# B&R Automation Studio project EFI (part 4)

### Cpu.per - X20CP1382/Cpu.per
```iecst
VAR_CONFIG
	gPermanentSN AT %M0; (*Serial Number of the machine*)
	gPermanentVersion AT %M100; (* *)
	gPermanentMachine AT %M148; (* *)
	gPermanentSwBelt AT %M500; (* *)
	gPermanentBlock AT %M600; (* *)
	gPermanentInksParSw AT %M800; (* *)
	gInksPermanentParBar AT %M2000; (* *)
	HoldingRegister AT %MW6000; (* *)
END_VAR
```

### @LIBRARY.LST - X20CP1382/EFI/@LIBRARY.LST
```
Library List, V30
FW;C:\BrAutomation\SafeDESIGNER 4.3\SafePROG\PLC\FW_LIB\PLCopen_SF;PLCopen_SF;3
FW;C:\BrAutomation\SafeDESIGNER 4.3\SafePROG\PLC\SafePCOS_31;SafePCOS_31;0
FW;C:\BrAutomation\SafeDESIGNER 4.3\SafePROG\PLC;IEC;3
```

### BusNavigator.iom - X20CP1382/EFI/BusNavigator.iom
```
IOOffsets (SIBytes=2048, SOBytes=2048, NSIBytes=1024, NSOBytes=1024, ConnectionsValidOffset=24, EMOsOffset=69, EMOsSize=64)
  Module SL1.SM1 (Hardware=X20SL8100, SafeLogicID=1, SafeModuleID=1, SISize=1, SOSize=1, NSISize=132, NSOSize=132, SIOffset=16, SOOffset=12, NSIOffset=0, NSOOffset=0, HWTypeCode=5)
    Channel ExternalMachineOption000 (Mapping=SIX69.0, Variable=SelectMachine)
    Channel BOOL001 (Mapping=NSQX0.0, Variable=g_xInputSelectMachine, SODIndex=0x2580, SODSubIndex=0x1)
    Channel INT001 (Mapping=NSQW2, Variable=ErrorCodeArea1, SODIndex=0x2580, SODSubIndex=0x2)
    Channel INT002 (Mapping=NSQW4, Variable=ErrorCodeArea2, SODIndex=0x2580, SODSubIndex=0x3)
  Module SL1.SM2 (Hardware=X20SC0402, SafeLogicID=1, SafeModuleID=2, SISize=4, SOSize=2, NSISize=1, NSOSize=1, SIOffset=20, SOOffset=16, NSIOffset=132, NSOOffset=132, ConnectionValidBitNumber=0, HWTypeCode=59)
    Channel SafeDigitalInput01 (Mapping=SIX20.0, Variable=InputReset, Address=Cyclic#1.::X20SLX402_006.DInput[1], SODIndex=0x6000, SODSubIndex=0x1)
    Channel SafeDigitalOutput01 (Mapping=SQX16.0, Variable=TransportEnable, SODIndex=0x6200, SODSubIndex=0x1)
    Channel ReleaseOutput01 (Mapping=NSQX132.0, Variable=ReleaseTransport, SODIndex=0x6200, SODSubIndex=0x2)
  Module SL1.SM3 (Hardware=X20SI8110, SafeLogicID=1, SafeModuleID=3, SISize=3, SOSize=0, NSISize=0, NSOSize=0, SIOffset=62, ConnectionValidBitNumber=1, HWTypeCode=27)
    Channel SafeDigitalInput01 (Mapping=SIX62.0, Variable=Rear01EStopBK1, Address=Cyclic#1.::X20SI8110_117.DInput[1], SODIndex=0x6000, SODSubIndex=0x1)
    Channel SafeDigitalInput02 (Mapping=SIX62.1, Variable=Rear02EStopBK1, Address=Cyclic#1.::X20SI8110_117.DInput[2], SODIndex=0x6000, SODSubIndex=0x1)
    Channel SafeDigitalInput03 (Mapping=SIX62.2, Variable=Front01EStopBK1, Address=Cyclic#1.::X20SI8110_117.DInput[3], SODIndex=0x6000, SODSubIndex=0x1)
    Channel SafeDigitalInput04 (Mapping=SIX62.3, Variable=Front02EStopBK1, Address=Cyclic#1.::X20SI8110_117.DInput[4], SODIndex=0x6000, SODSubIndex=0x1)
    Channel SafeDigitalInput05 (Mapping=SIX62.4, Variable=LightCurtain01BK1, Address=Cyclic#1.::X20SI8110_117.DInput[5], SODIndex=0x6000, SODSubIndex=0x1)
    Channel SafeDigitalInput06 (Mapping=SIX62.5, Variable=GuardSwitchBK1, Address=Cyclic#1.::X20SI8110_117.DInput[6], SODIndex=0x6000, SODSubIndex=0x1)
    Channel SafeDigitalInput07 (Mapping=SIX62.6, Variable=LightCurtain02BK1, Address=Cyclic#1.::X20SI8110_117.DInput[7], SODIndex=0x6000, SODSubIndex=0x1)
  Module SL1.SM4 (Hardware=X20SO2110, SafeLogicID=1, SafeModuleID=4, SISize=1, SOSize=1, NSISize=1, NSOSize=1, SIOffset=61, SOOffset=14, NSIOffset=133, NSOOffset=133, ConnectionValidBitNumber=2, HWTypeCode=43)
    Channel SafeDigitalOutput01 (Mapping=SQX14.0, Variable=UpDownBK1Enable, SODIndex=0x6200, SODSubIndex=0x1)
    Channel SafeDigitalOutput02 (Mapping=SQX14.1, Variable=IclaBK1Enable, SODIndex=0x6200, SODSubIndex=0x1)
    Channel ReleaseOutput01 (Mapping=NSQX133.0, Variable=ReleaseUpDownBK1, SODIndex=0x6200, SODSubIndex=0x2)
    Channel ReleaseOutput02 (Mapping=NSQX133.1, Variable=ReleaseIclaBK1, SODIndex=0x6200, SODSubIndex=0x2)
  Module SL1.SM5 (Hardware=X20SI8110, SafeLogicID=1, SafeModuleID=5, SISize=3, SOSize=0, NSISize=0, NSOSize=0, SIOffset=66, ConnectionValidBitNumber=3, HWTypeCode=27)
    Channel SafeDigitalInput01 (Mapping=SIX66.0, Variable=Rear01EStopBK2, Address=Cyclic#1.::X20SI8110_217.DInput[1], SODIndex=0x6000, SODSubIndex=0x1)
    Channel SafeDigitalInput02 (Mapping=SIX66.1, Variable=Rear02EStopBK2, Address=Cyclic#1.::X20SI8110_217.DInput[2], SODIndex=0x6000, SODSubIndex=0x1)
    Channel SafeDigitalInput03 (Mapping=SIX66.2, Variable=Front01EStopBK2, Address=Cyclic#1.::X20SI8110_217.DInput[3], SODIndex=0x6000, SODSubIndex=0x1)
    Channel SafeDigitalInput04 (Mapping=SIX66.3, Variable=Front02EStopBK2, Address=Cyclic#1.::X20SI8110_217.DInput[4], SODIndex=0x6000, SODSubIndex=0x1)
    Channel SafeDigitalInput05 (Mapping=SIX66.4, Variable=LightCurtain01BK2, Address=Cyclic#1.::X20SI8110_217.DInput[5], SODIndex=0x6000, SODSubIndex=0x1)
    Channel SafeDigitalInput06 (Mapping=SIX66.5, Variable=GuardSwitchBK2, Address=Cyclic#1.::X20SI8110_217.DInput[6], SODIndex=0x6000, SODSubIndex=0x1)
    Channel SafeDigitalInput07 (Mapping=SIX66.6, Variable=LightCurtain02BK2, Address=Cyclic#1.::X20SI8110_217.DInput[7], SODIndex=0x6000, SODSubIndex=0x1)
  Module SL1.SM6 (Hardware=X20SO2110, SafeLogicID=1, SafeModuleID=6, SISize=1, SOSize=1, NSISize=1, NSOSize=1, SIOffset=65, SOOffset=15, NSIOffset=134, NSOOffset=134, ConnectionValidBitNumber=4, HWTypeCode=43)
    Channel SafeDigitalOutput01 (Mapping=SQX15.0, Variable=UpDownBK2Enable, SODIndex=0x6200, SODSubIndex=0x1)
    Channel SafeDigitalOutput02 (Mapping=SQX15.1, Variable=IclaBK2Enable, SODIndex=0x6200, SODSubIndex=0x1)
    Channel ReleaseOutput01 (Mapping=NSQX134.0, Variable=ReleaseUpDownBK2, SODIndex=0x6200, SODSubIndex=0x2)
    Channel ReleaseOutput02 (Mapping=NSQX134.1, Variable=ReleaseIclaBK2, SODIndex=0x6200, SODSubIndex=0x2)
```

### CHGUNITS.LST - X20CP1382/EFI/CHGUNITS.LST
```
(*
NPOU: 2
*)
PG	Main
FB	MOVE_UINT
```

### CROSSREF.CSV - X20CP1382/EFI/CROSSREF.CSV
```
C000,POE\Main\Code.GB,4,IN,282,90,Read,,INT,,,VAR_GLOBAL,GLOBAL,,
C000,POE\Main\Code.GB,5,IN,283,55,Read,,INT,,,VAR_GLOBAL,GLOBAL,,
C000,POE\Main\Code.GB,8,IN,287,58,Read,,INT,,,VAR_GLOBAL,GLOBAL,,
C000,POE\Main\Code.GB,8,IN,289,0,Read,,INT,,,VAR_GLOBAL,GLOBAL,,
C000,POE\Main\Code.GB,8,IN,285,39,Read,,INT,,,VAR_GLOBAL,GLOBAL,,
C000,POE\Main\Code.GB,19,IN,421,84,Read,,INT,,,VAR_GLOBAL,GLOBAL,,
C000,POE\Main\Code.GB,20,IN,437,54,Read,,INT,,,VAR_GLOBAL,GLOBAL,,
C000,POE\Main\Code.GB,22,IN,571,82,Read,,INT,,,VAR_GLOBAL,GLOBAL,,
C000,POE\Main\Code.GB,23,IN,493,38,Read,,INT,,,VAR_GLOBAL,GLOBAL,,
C000,POE\Main\Code.GB,23,IN,604,48,Read,,INT,,,VAR_GLOBAL,GLOBAL,,
ErrorCodeArea1,POE\Main\Code.GB,11,OUT,307,71,Write,,INT,NSQW2,,VAR_GLOBAL,GLOBAL,,
ErrorCodeArea2,POE\Main\Code.GB,26,OUT,800,82,Write,,INT,NSQW4,,VAR_GLOBAL,GLOBAL,,
Front01EStopBK1,POE\Main\Code.GB,1,IN,310,8,Read,,SAFEBOOL,SIX62.2,,VAR_GLOBAL,GLOBAL,,
Front01EStopBK2,POE\Main\Code.GB,16,IN,392,8,Read,,SAFEBOOL,SIX66.2,,VAR_GLOBAL,GLOBAL,,
Front02EStopBK1,POE\Main\Code.GB,1,IN,311,8,Read,,SAFEBOOL,SIX62.3,,VAR_GLOBAL,GLOBAL,,
Front02EStopBK2,POE\Main\Code.GB,16,IN,393,8,Read,,SAFEBOOL,SIX66.3,,VAR_GLOBAL,GLOBAL,,
g_xInputSelectMachine,POE\Main\Code.GB,16,OUT,855,37,Write,,BOOL,NSQX0.0,,VAR_GLOBAL,GLOBAL,,
GuardSwitchBK1,POE\Main\Code.GB,4,IN,312,23,Read,,SAFEBOOL,SIX62.5,,VAR_GLOBAL,GLOBAL,,
GuardSwitchBK2,POE\Main\Code.GB,19,IN,477,47,Read,,SAFEBOOL,SIX66.5,,VAR_GLOBAL,GLOBAL,,
IclaBK1Enable,POE\Main\Code.GB,29,OUT,769,81,Write,,SAFEBOOL,SQX14.1,,VAR_GLOBAL,GLOBAL,,
IclaBK2Enable,POE\Main\Code.GB,32,OUT,683,77,Write,,SAFEBOOL,SQX15.1,,VAR_GLOBAL,GLOBAL,,
InputReset,POE\Main\Code.GB,1,IN,37,83,Read,,SAFEBOOL,SIX20.0,,VAR_GLOBAL,GLOBAL,,
InputReset,POE\Main\Code.GB,2,IN,27,0,Read,,SAFEBOOL,SIX20.0,,VAR_GLOBAL,GLOBAL,,
InputReset,POE\Main\Code.GB,7,IN,155,47,Read,,SAFEBOOL,SIX20.0,,VAR_GLOBAL,GLOBAL,,
InputReset,POE\Main\Code.GB,8,IN,211,0,Read,,SAFEBOOL,SIX20.0,,VAR_GLOBAL,GLOBAL,,
InputReset,POE\Main\Code.GB,17,IN,362,30,Read,,SAFEBOOL,SIX20.0,,VAR_GLOBAL,GLOBAL,,
InputReset,POE\Main\Code.GB,20,IN,390,0,Read,,SAFEBOOL,SIX20.0,,VAR_GLOBAL,GLOBAL,,
InputReset,POE\Main\Code.GB,22,IN,547,81,Read,,SAFEBOOL,SIX20.0,,VAR_GLOBAL,GLOBAL,,
InputReset,POE\Main\Code.GB,22,IN,475,58,Read,,SAFEBOOL,SIX20.0,,VAR_GLOBAL,GLOBAL,,
InputReset,POE\Main\Code.GB,29,IN,774,15,Read,,SAFEBOOL,SIX20.0,,VAR_GLOBAL,GLOBAL,,
InputReset,POE\Main\Code.GB,29,IN,718,6,Read,,SAFEBOOL,SIX20.0,,VAR_GLOBAL,GLOBAL,,
InputReset,POE\Main\Code.GB,32,IN,652,23,Read,,SAFEBOOL,SIX20.0,,VAR_GLOBAL,GLOBAL,,
LightCurtain01BK1,POE\Main\Code.GB,7,IN,317,10,Read,,SAFEBOOL,SIX62.4,,VAR_GLOBAL,GLOBAL,,
LightCurtain01BK2,POE\Main\Code.GB,22,IN,549,3,Read,,SAFEBOOL,SIX66.4,,VAR_GLOBAL,GLOBAL,,
LightCurtain02BK1,POE\Main\Code.GB,7,IN,318,9,Read,,SAFEBOOL,SIX62.6,,VAR_GLOBAL,GLOBAL,,
LightCurtain02BK2,POE\Main\Code.GB,22,IN,559,3,Read,,SAFEBOOL,SIX66.6,,VAR_GLOBAL,GLOBAL,,
Rear01EStopBK1,POE\Main\Code.GB,1,IN,308,13,Read,,SAFEBOOL,SIX62.0,,VAR_GLOBAL,GLOBAL,,
Rear01EStopBK2,POE\Main\Code.GB,16,IN,394,49,Read,,SAFEBOOL,SIX66.0,,VAR_GLOBAL,GLOBAL,,
Rear02EStopBK1,POE\Main\Code.GB,1,IN,309,13,Read,,SAFEBOOL,SIX62.1,,VAR_GLOBAL,GLOBAL,,
Rear02EStopBK2,POE\Main\Code.GB,16,IN,395,49,Read,,SAFEBOOL,SIX66.1,,VAR_GLOBAL,GLOBAL,,
ReleaseIclaBK1,POE\Main\Code.GB,30,OUT,773,78,Write,,BOOL,NSQX133.1,,VAR_GLOBAL,GLOBAL,,
ReleaseIclaBK2,POE\Main\Code.GB,33,OUT,689,81,Write,,BOOL,NSQX134.1,,VAR_GLOBAL,GLOBAL,,
ReleaseTransport,POE\Main\Code.GB,27,OUT,719,66,Write,,BOOL,NSQX132.0,,VAR_GLOBAL,GLOBAL,,
ReleaseUpDownBK1,POE\Main\Code.GB,30,OUT,772,74,Write,,BOOL,NSQX133.0,,VAR_GLOBAL,GLOBAL,,
ReleaseUpDownBK2,POE\Main\Code.GB,33,OUT,688,77,Write,,BOOL,NSQX134.0,,VAR_GLOBAL,GLOBAL,,
SelectMachine,POE\Main\Code.GB,16,IN,801,53,Read,,SAFEBOOL,SIX69.0,,VAR_GLOBAL,GLOBAL,,
SelectMachine,POE\Main\Code.GB,16,IN,804,12,Read,,SAFEBOOL,SIX69.0,,VAR_GLOBAL,GLOBAL,,
SelectMachine,POE\Main\Code.GB,16,IN,856,10,Read,,SAFEBOOL,SIX69.0,,VAR_GLOBAL,GLOBAL,,
SelectMachine,POE\Main\Code.GB,17,IN,802,29,Read,,SAFEBOOL,SIX69.0,,VAR_GLOBAL,GLOBAL,,
SelectMachine,POE\Main\Code.GB,17,IN,803,0,Read,,SAFEBOOL,SIX69.0,,VAR_GLOBAL,GLOBAL,,
SelectMachine,POE\Main\Code.GB,19,IN,805,57,Read,,SAFEBOOL,SIX69.0,,VAR_GLOBAL,GLOBAL,,
SelectMachine,POE\Main\Code.GB,22,IN,806,8,Read,,SAFEBOOL,SIX69.0,,VAR_GLOBAL,GLOBAL,,
SelectMachine,POE\Main\Code.GB,22,IN,807,80,Read,,SAFEBOOL,SIX69.0,,VAR_GLOBAL,GLOBAL,,
SelectMachine,POE\Main\Code.GB,25,IN,812,23,Read,,SAFEBOOL,SIX69.0,,VAR_GLOBAL,GLOBAL,,
SelectMachine,POE\Main\Code.GB,28,IN,835,5,Read,,SAFEBOOL,SIX69.0,,VAR_GLOBAL,GLOBAL,,
TransportEnable,POE\Main\Code.GB,25,OUT,716,0,Write,,SAFEBOOL,SQX16.0,,VAR_GLOBAL,GLOBAL,,
TransportEnable,POE\Main\Code.GB,28,IN,770,44,Read,,SAFEBOOL,SQX16.0,,VAR_GLOBAL,GLOBAL,,
TransportEnable,POE\Main\Code.GB,28,IN,649,64,Read,,SAFEBOOL,SQX16.0,,VAR_GLOBAL,GLOBAL,,
UpDownBK1Enable,POE\Main\Code.GB,29,OUT,768,78,Write,,SAFEBOOL,SQX14.0,,VAR_GLOBAL,GLOBAL,,
UpDownBK2Enable,POE\Main\Code.GB,29,OUT,682,74,Write,,SAFEBOOL,SQX15.0,,VAR_GLOBAL,GLOBAL,,
```

### EFI.proj - X20CP1382/EFI/EFI/EFI/EFI.proj
```
Project (DefaultTargets=Build, ToolsVersion=2.0)
  Import (Project=$(AdeProjectTargetsPath), Condition='$(AdeProjectTargetsPath)' != '')
  PropertyGroup:
    ProjectName = EFI
    AdeProductVersion = 1.0.0.0
  ItemGroup:
    AdditionalCompareData (Include=Hardware\AdditionalCompareResults.txc)
  ItemGroup:
    Folder (Include=References)
      FolderType = References
      Visible = false
    Folder (Include=Libraries)
      FolderType = Root
    Folder (Include=Logical Elements)
      FolderType = Root
      DisplayName = Logical POUs
    Folder (Include=Hardware)
      FolderType = Root
      Visible = false
    Folder (Include=Hardware\PLC)
      FolderType = Configuration
    Folder (Include=Hardware\PLC\CPU)
      FolderType = Resource
  ItemGroup:
    IoConfigurationWorksheet (Include=Hardware\PLC\CPU\IO_Configuration.ioc)
  ItemGroup:
    ProgramOrganizationUnit (Include=Logical Elements\Main.pou)
    ProgramOrganizationUnit (Include=Logical Elements\MOVE_UINT.pou)
  ItemGroup:
    ResourceSettings (Include=Hardware\PLC\CPU\ResourceSettings.set)
      DisplayName = Tasks
  ItemGroup:
    SolutionReference (Include=PLCopen_SF)
  ItemGroup:
    VariableWorksheet (Include=Hardware\PLC\CPU\Exchange_Variables.var)
    VariableWorksheet (Include=Hardware\PLC\CPU\Global_Variables.var)
    VariableWorksheet (Include=Hardware\PLC\CPU\AutoGenerated_VarConfig.var)
      IsVarConfig = true
      AutoGenerated = true
```

### Global_Variables.var - X20CP1382/EFI/EFI/EFI/Hardware/PLC/CPU/Global_Variables.var
```iecst
{GroupDefinition(0,'NewGroup')}

VAR_GLOBAL {Group(0)}
    {LINE(1)}
    C000 : INT := -16384;
    {LINE(2)}
    ErrorCodeArea1 AT %QW2 : INT {Custom('SL1.SM1.INT001')};
    {LINE(3)}
    Rear01EStopBK1 AT %IX62.0 : SAFEBOOL {SafeAdr(true),Custom('SL1.SM3.SafeDigitalInput01')};
    {LINE(4)}
    Rear02EStopBK1 AT %IX62.1 : SAFEBOOL {SafeAdr(true),Custom('SL1.SM3.SafeDigitalInput02')};
    {LINE(5)}
    Front01EStopBK1 AT %IX62.2 : SAFEBOOL {SafeAdr(true),Custom('SL1.SM3.SafeDigitalInput03')};
    {LINE(6)}
    Front02EStopBK1 AT %IX62.3 : SAFEBOOL {SafeAdr(true),Custom('SL1.SM3.SafeDigitalInput04')};
    {LINE(7)}
    GuardSwitchBK1 AT %IX62.5 : SAFEBOOL {SafeAdr(true),Custom('SL1.SM3.SafeDigitalInput06')};
    {LINE(8)}
    LightCurtain01BK1 AT %IX62.4 : SAFEBOOL {SafeAdr(true),Custom('SL1.SM3.SafeDigitalInput05')};
    {LINE(9)}
    LightCurtain02BK1 AT %IX62.6 : SAFEBOOL {SafeAdr(true),Custom('SL1.SM3.SafeDigitalInput07')};
    {LINE(10)}
    UpDownBK1Enable AT %QX14.0 : SAFEBOOL {SafeAdr(true),Custom('SL1.SM4.SafeDigitalOutput01')};
    {LINE(11)}
    IclaBK1Enable AT %QX14.1 : SAFEBOOL {SafeAdr(true),Custom('SL1.SM4.SafeDigitalOutput02')};
    {LINE(12)}
    TransportEnable AT %QX16.0 : SAFEBOOL {SafeAdr(true),Custom('SL1.SM2.SafeDigitalOutput01')};
    {LINE(13)}
    InputReset AT %IX20.0 : SAFEBOOL {SafeAdr(true),Custom('SL1.SM2.SafeDigitalInput01')};
    {LINE(14)}
    ReleaseTransport AT %QX132.0 : BOOL {Custom('SL1.SM2.ReleaseOutput01')};
    {LINE(15)}
    ReleaseUpDownBK1 AT %QX133.0 : BOOL {Custom('SL1.SM4.ReleaseOutput01')};
    {LINE(16)}
    ReleaseIclaBK1 AT %QX133.1 : BOOL {Custom('SL1.SM4.ReleaseOutput02')};
    {LINE(17)}
    Front01EStopBK2 AT %IX66.2 : SAFEBOOL {SafeAdr(true),Custom('SL1.SM5.SafeDigitalInput03')};
    {LINE(18)}
    Front02EStopBK2 AT %IX66.3 : SAFEBOOL {SafeAdr(true),Custom('SL1.SM5.SafeDigitalInput04')};
    {LINE(19)}
    Rear01EStopBK2 AT %IX66.0 : SAFEBOOL {SafeAdr(true),Custom('SL1.SM5.SafeDigitalInput01')};
    {LINE(20)}
    Rear02EStopBK2 AT %IX66.1 : SAFEBOOL {SafeAdr(true),Custom('SL1.SM5.SafeDigitalInput02')};
    {LINE(21)}
    GuardSwitchBK2 AT %IX66.5 : SAFEBOOL {SafeAdr(true),Custom('SL1.SM5.SafeDigitalInput06')};
    {LINE(22)}
    LightCurtain01BK2 AT %IX66.4 : SAFEBOOL {SafeAdr(true),Custom('SL1.SM5.SafeDigitalInput05')};
    {LINE(23)}
    LightCurtain02BK2 AT %IX66.6 : SAFEBOOL {SafeAdr(true),Custom('SL1.SM5.SafeDigitalInput07')};
    {LINE(24)}
    UpDownBK2Enable AT %QX15.0 : SAFEBOOL {SafeAdr(true),Custom('SL1.SM6.SafeDigitalOutput01')};
    {LINE(25)}
    IclaBK2Enable AT %QX15.1 : SAFEBOOL {SafeAdr(true),Custom('SL1.SM6.SafeDigitalOutput02')};
    {LINE(26)}
    ReleaseUpDownBK2 AT %QX134.0 : BOOL {Custom('SL1.SM6.ReleaseOutput01')};
    {LINE(27)}
    ReleaseIclaBK2 AT %QX134.1 : BOOL {Custom('SL1.SM6.ReleaseOutput02')};
    {LINE(28)}
    ErrorCodeArea2 AT %QW4 : INT {Custom('SL1.SM1.INT002')};
    {LINE(29)}
    SelectMachine AT %IX69.0 : SAFEBOOL {SafeAdr(true),Custom('SL1.SM1.ExternalMachineOption000')};
    {LINE(30)}
    g_xInputSelectMachine AT %QX0.0 : BOOL {Custom('SL1.SM1.BOOL001')};
END_VAR
```

### PROJECT.INF - X20CP1382/EFI/PROJECT.INF
```
[@_ProjInfo_@]
LastChange=04/04/2019  12:03:54
[SDIO]
Worksheet.Crc=0x20128ECF
[ProjectAccess]
DEVELOPMENT=25D55AD283AA400AF464C76D713C07AD
COMMISSIONING=E10ADC3949BA59ABBE56E057F20F883E
[UserInterface]
AccessTimeOut=3600000
```

### IoMap.iom - X20CP1382/IoMap.iom
```iecst
VAR_CONFIG
	Cyclic#4.::X20DOF322_001.DOutput[1] AT %QX."X20DOF322_001".DigitalOutput01;
	Cyclic#4.::X20DOF322_001.DOutput[16] AT %QX."X20DOF322_001".DigitalOutput16;
	Cyclic#4.::X20DOF322_001.DOutput[2] AT %QX."X20DOF322_001".DigitalOutput02;
	Cyclic#4.::X20DOF322_001.DOutput[3] AT %QX."X20DOF322_001".DigitalOutput03;
	Cyclic#4.::X20DOF322_001.DOutput[4] AT %QX."X20DOF322_001".DigitalOutput04;
	Cyclic#4.::X20DOF322_001.DOutput[5] AT %QX."X20DOF322_001".DigitalOutput05;
	Cyclic#4.::X20DOF322_001.DOutput[6] AT %QX."X20DOF322_001".DigitalOutput06;
	Cyclic#4.::X20DOF322_001.DOutput[7] AT %QX."X20DOF322_001".DigitalOutput07;
	Cyclic#4.::X20DOF322_001.DOutput[8] AT %QX."X20DOF322_001".DigitalOutput08;
	Cyclic#4.::X20DOF322_001.DOutput[9] AT %QX."X20DOF322_001".DigitalOutput09;
	Cyclic#4.::X20DOF322_001.DOutput[10] AT %QX."X20DOF322_001".DigitalOutput10;
	Cyclic#4.::X20DOF322_001.DOutput[11] AT %QX."X20DOF322_001".DigitalOutput11;
	Cyclic#4.::X20DOF322_001.DOutput[12] AT %QX."X20DOF322_001".DigitalOutput12;
	Cyclic#4.::X20DOF322_001.DOutput[13] AT %QX."X20DOF322_001".DigitalOutput13;
	Cyclic#4.::X20DOF322_001.DOutput[14] AT %QX."X20DOF322_001".DigitalOutput14;
	Cyclic#4.::X20DOF322_001.DOutput[15] AT %QX."X20DOF322_001".DigitalOutput15;
	Cyclic#4.::X20DIF371_002.DInput[1] AT %IX."X20DIF371_002".DigitalInput01;
	Cyclic#4.::X20DIF371_002.DInput[2] AT %IX."X20DIF371_002".DigitalInput02;
	Cyclic#4.::X20DIF371_002.DInput[3] AT %IX."X20DIF371_002".DigitalInput03;
	Cyclic#4.::X20DIF371_002.DInput[4] AT %IX."X20DIF371_002".DigitalInput04;
	Cyclic#4.::X20DIF371_002.DInput[5] AT %IX."X20DIF371_002".DigitalInput05;
	Cyclic#4.::X20DIF371_002.DInput[6] AT %IX."X20DIF371_002".DigitalInput06;
	Cyclic#4.::X20DIF371_002.DInput[7] AT %IX."X20DIF371_002".DigitalInput07;
	Cyclic#4.::X20DIF371_002.DInput[8] AT %IX."X20DIF371_002".DigitalInput08;
	Cyclic#4.::X20DIF371_002.DInput[9] AT %IX."X20DIF371_002".DigitalInput09;
	Cyclic#4.::X20DIF371_002.DInput[10] AT %IX."X20DIF371_002".DigitalInput10;
	Cyclic#4.::X20DIF371_002.DInput[11] AT %IX."X20DIF371_002".DigitalInput11;
	Cyclic#4.::X20DIF371_002.DInput[12] AT %IX."X20DIF371_002".DigitalInput12;
	Cyclic#4.::X20DIF371_002.DInput[13] AT %IX."X20DIF371_002".DigitalInput13;
	Cyclic#4.::X20DIF371_002.DInput[14] AT %IX."X20DIF371_002".DigitalInput14;
	Cyclic#4.::X20DIF371_002.DInput[15] AT %IX."X20DIF371_002".DigitalInput15;
	Cyclic#4.::X20DIF371_002.DInput[16] AT %IX."X20DIF371_002".DigitalInput16;
	Cyclic#4.::X20DOF322_001.ModuleOk AT %IX."X20DOF322_001".ModuleOk;
	Cyclic#4.::X1.DInput[1] AT %IX."X1".DigitalInput01;
	Cyclic#4.::X1.DInput[2] AT %IX."X1".DigitalInput02;
	Cyclic#4.::X1.DInput[3] AT %IX."X1".DigitalInput03;
	Cyclic#4.::X1.DInput[4] AT %IX."X1".DigitalInput04;
	Cyclic#4.::X1.AInput[1] AT %IW."X1".AnalogInput01;
	Cyclic#4.::X1.AInput[2] AT %IW."X1".AnalogInput02;
	Cyclic#4.::X1.Status01 AT %IB."X1".StatusInput01;
	Cyclic#4.::X2.DInput[1] AT %IX."X2".DigitalInput01;
	Cyclic#4.::X2.DInput[2] AT %IX."X2".DigitalInput02;
	Cyclic#4.::X2.DInput[3] AT %IX."X2".DigitalInput03;
	Cyclic#4.::X2.DInput[4] AT %IX."X2".DigitalInput04;
	Cyclic#4.::X2.DInput[5] AT %IX."X2".DigitalInput05;
	Cyclic#4.::X2.DInput[6] AT %IX."X2".DigitalInput06;
	Cyclic#4.::X2.DInput[7] AT %IX."X2".DigitalInput07;
	Cyclic#4.::X2.DInput[8] AT %IX."X2".DigitalInput08;
	Cyclic#4.::X2.DInput[9] AT %IX."X2".DigitalInput09;
	Cyclic#4.::X2.DInput[10] AT %IX."X2".DigitalInput10;
	Cyclic#2.::X2.DInput[11] AT %IX."X2".DigitalInput11;
	Cyclic#2.::X2.DInput[12] AT %IX."X2".DigitalInput12;
	Cyclic#2.::X2.DInput[13] AT %IX."X2".DigitalInput13;
	Cyclic#4.::X2.DInput[14] AT %IX."X2".DigitalInput14;
	Cyclic#4.::X20DIF371_002.ModuleOk AT %IX."X20DIF371_002".ModuleOk;
	Cyclic#4.::X20DIF371_003.DInput[1] AT %IX."X20DIF371_003".DigitalInput01;
	Cyclic#4.::X20DIF371_003.DInput[2] AT %IX."X20DIF371_003".DigitalInput02;
	Cyclic#4.::X20DIF371_003.DInput[3] AT %IX."X20DIF371_003".DigitalInput03;
	Cyclic#4.::X20DIF371_003.DInput[4] AT %IX."X20DIF371_003".DigitalInput04;
	Cyclic#4.::X20DIF371_003.DInput[5] AT %IX."X20DIF371_003".DigitalInput05;
	Cyclic#4.::X20DIF371_003.DInput[6] AT %IX."X20DIF371_003".DigitalInput06;
	Cyclic#4.::X20DIF371_003.DInput[7] AT %IX."X20DIF371_003".DigitalInput07;
	Cyclic#4.::X20DIF371_003.DInput[8] AT %IX."X20DIF371_003".DigitalInput08;
	Cyclic#4.::X20DIF371_003.DInput[9] AT %IX."X20DIF371_003".DigitalInput09;
	Cyclic#4.::X20DIF371_003.DInput[10] AT %IX."X20DIF371_003".DigitalInput10;
	Cyclic#4.::X20DIF371_003.DInput[11] AT %IX."X20DIF371_003".DigitalInput11;
	Cyclic#4.::X20DIF371_003.DInput[12] AT %IX."X20DIF371_003".DigitalInput12;
	Cyclic#4.::X20DIF371_003.DInput[13] AT %IX."X20DIF371_003".DigitalInput13;
	Cyclic#4.::X20DIF371_003.DInput[14] AT %IX."X20DIF371_003".DigitalInput14;
	Cyclic#4.::X20DIF371_003.DInput[15] AT %IX."X20DIF371_003".DigitalInput15;
	Cyclic#4.::X20DIF371_003.DInput[16] AT %IX."X20DIF371_003".DigitalInput16;
	Cyclic#4.::X20DOF322_004.DOutput[1] AT %QX."X20DOF322_004".DigitalOutput01;
	Cyclic#4.::X20DOF322_004.DOutput[2] AT %QX."X20DOF322_004".DigitalOutput02;
	Cyclic#4.::X20DOF322_004.DOutput[3] AT %QX."X20DOF322_004".DigitalOutput03;
	Cyclic#4.::X20DOF322_004.DOutput[4] AT %QX."X20DOF322_004".DigitalOutput04;
	Cyclic#4.::X20DOF322_004.DOutput[5] AT %QX."X20DOF322_004".DigitalOutput05;
	Cyclic#4.::X20DOF322_004.DOutput[6] AT %QX."X20DOF322_004".DigitalOutput06;
	Cyclic#4.::X20DOF322_004.DOutput[7] AT %QX."X20DOF322_004".DigitalOutput07;
	Cyclic#4.::X20DOF322_004.DOutput[8] AT %QX."X20DOF322_004".DigitalOutput08;
	Cyclic#4.::X20DOF322_004.DOutput[9] AT %QX."X20DOF322_004".DigitalOutput09;
	Cyclic#4.::X20DOF322_004.DOutput[10] AT %QX."X20DOF322_004".DigitalOutput10;
	Cyclic#4.::X20DOF322_004.DOutput[11] AT %QX."X20DOF322_004".DigitalOutput11;
	Cyclic#4.::X20DOF322_004.DOutput[12] AT %QX."X20DOF322_004".DigitalOutput12;
	Cyclic#4.::X20DOF322_004.DOutput[13] AT %QX."X20DOF322_004".DigitalOutput13;
	Cyclic#4.::X20DOF322_004.DOutput[14] AT %QX."X20DOF322_004".DigitalOutput14;
	Cyclic#4.::X20DOF322_004.DOutput[15] AT %QX."X20DOF322_004".DigitalOutput15;
	Cyclic#4.::X20DOF322_004.DOutput[16] AT %QX."X20DOF322_004".DigitalOutput16;
	Cyclic#4.::X20DOF322_004.ModuleOk AT %IX."X20DOF322_004".ModuleOk;
	Cyclic#4.::X20DIF371_101.DInput[1] AT %IX."X20DIF371_101".DigitalInput01;
	Cyclic#4.::X20DIF371_101.DInput[2] AT %IX."X20DIF371_101".DigitalInput02;
	Cyclic#4.::X20DIF371_101.DInput[3] AT %IX."X20DIF371_101".DigitalInput03;
	Cyclic#4.::X20DIF371_101.DInput[4] AT %IX."X20DIF371_101".DigitalInput04;
	Cyclic#4.::X20DIF371_101.DInput[5] AT %IX."X20DIF371_101".DigitalInput05;
	Cyclic#4.::X20DIF371_101.DInput[6] AT %IX."X20DIF371_101".DigitalInput06;
	Cyclic#4.::X20DIF371_101.DInput[7] AT %IX."X20DIF371_101".DigitalInput07;
	Cyclic#4.::X20DIF371_101.DInput[8] AT %IX."X20DIF371_101".DigitalInput08;
	Cyclic#4.::X20DIF371_101.DInput[9] AT %IX."X20DIF371_101".DigitalInput09;
	Cyclic#4.::X20DIF371_101.DInput[10] AT %IX."X20DIF371_101".DigitalInput10;
	Cyclic#4.::X20DIF371_101.DInput[11] AT %IX."X20DIF371_101".DigitalInput11;
	Cyclic#4.::X20DIF371_101.DInput[12] AT %IX."X20DIF371_101".DigitalInput12;
	Cyclic#4.::X20DIF371_101.DInput[13] AT %IX."X20DIF371_101".DigitalInput13;
	Cyclic#4.::X20DIF371_101.DInput[14] AT %IX."X20DIF371_101".DigitalInput14;
	Cyclic#4.::X20DIF371_101.DInput[15] AT %IX."X20DIF371_101".DigitalInput15;
	Cyclic#4.::X20DIF371_101.DInput[16] AT %IX."X20DIF371_101".DigitalInput16;
	Cyclic#4.::X20DIF371_102.DInput[1] AT %IX."X20DIF371_102".DigitalInput01;
	Cyclic#4.::X20DIF371_102.DInput[2] AT %IX."X20DIF371_102".DigitalInput02;
	Cyclic#4.::X20DIF371_102.DInput[3] AT %IX."X20DIF371_102".DigitalInput03;
	Cyclic#4.::X20DIF371_102.DInput[4] AT %IX."X20DIF371_102".DigitalInput04;
	Cyclic#4.::X20DIF371_102.DInput[5] AT %IX."X20DIF371_102".DigitalInput05;
	Cyclic#4.::X20DIF371_102.DInput[6] AT %IX."X20DIF371_102".DigitalInput06;
	Cyclic#4.::X20DIF371_102.DInput[7] AT %IX."X20DIF371_102".DigitalInput07;
	Cyclic#4.::X20DIF371_102.DInput[8] AT %IX."X20DIF371_102".DigitalInput08;
	Cyclic#4.::X20DIF371_102.DInput[9] AT %IX."X20DIF371_102".DigitalInput09;
	Cyclic#4.::X20DIF371_102.DInput[10] AT %IX."X20DIF371_102".DigitalInput10;
	Cyclic#4.::X20DIF371_102.DInput[11] AT %IX."X20DIF371_102".DigitalInput11;
	Cyclic#4.::X20DIF371_102.DInput[12] AT %IX."X20DIF371_102".DigitalInput12;
	Cyclic#4.::X20DIF371_102.DInput[13] AT %IX."X20DIF371_102".DigitalInput13;
	Cyclic#4.::X20DIF371_102.DInput[14] AT %IX."X20DIF371_102".DigitalInput14;
	Cyclic#4.::X20DIF371_102.DInput[15] AT %IX."X20DIF371_102".DigitalInput15;
	Cyclic#4.::X20DIF371_102.DInput[16] AT %IX."X20DIF371_102".DigitalInput16;
	Cyclic#4.::X20DIF371_103.DInput[1] AT %IX."X20DIF371_103".DigitalInput01;
	Cyclic#4.::X20DIF371_103.DInput[2] AT %IX."X20DIF371_103".DigitalInput02;
	Cyclic#4.::X20DIF371_103.DInput[3] AT %IX."X20DIF371_103".DigitalInput03;
	Cyclic#4.::X20DIF371_103.DInput[4] AT %IX."X20DIF371_103".DigitalInput04;
	Cyclic#4.::X20DIF371_103.DInput[5] AT %IX."X20DIF371_103".DigitalInput05;
	Cyclic#4.::X20DIF371_103.DInput[6] AT %IX."X20DIF371_103".DigitalInput06;
	Cyclic#4.::X20DIF371_103.DInput[7] AT %IX."X20DIF371_103".DigitalInput07;
	Cyclic#4.::X20DIF371_103.DInput[8] AT %IX."X20DIF371_103".DigitalInput08;
	Cyclic#4.::X20DIF371_103.DInput[9] AT %IX."X20DIF371_103".DigitalInput09;
	Cyclic#4.::X20DIF371_103.DInput[10] AT %IX."X20DIF371_103".DigitalInput10;
	Cyclic#4.::X20DIF371_103.DInput[11] AT %IX."X20DIF371_103".DigitalInput11;
	Cyclic#4.::X20DIF371_103.DInput[12] AT %IX."X20DIF371_103".DigitalInput12;
	Cyclic#4.::X20DIF371_103.DInput[13] AT %IX."X20DIF371_103".DigitalInput13;
	Cyclic#4.::X20DIF371_103.DInput[14] AT %IX."X20DIF371_103".DigitalInput14;
	Cyclic#4.::X20DIF371_103.DInput[15] AT %IX."X20DIF371_103".DigitalInput15;
	Cyclic#4.::X20DIF371_103.DInput[16] AT %IX."X20DIF371_103".DigitalInput16;
	Cyclic#4.::X20DIF371_101.ModuleOk AT %IX."X20DIF371_101".ModuleOk;
	Cyclic#4.::X20DIF371_102.ModuleOk AT %IX."X20DIF371_102".ModuleOk;
	Cyclic#4.::X20DIF371_103.ModuleOk AT %IX."X20DIF371_103".ModuleOk;
	Cyclic#4.::X20AI8321_109.AInput[1] AT %IW."X20AI8321_109".AnalogInput01; (*Current 0 to 20 mA / current 4 to 20 mA ; P4 is working with current 4 to 20 mA, resolution 12 bit*)
	Cyclic#4.::X20AI8321_109.AInput[2] AT %IW."X20AI8321_109".AnalogInput02; (*Current 0 to 20 mA / current 4 to 20 mA ; P4 is working with current 4 to 20 mA, resolution 12 bit*)
	Cyclic#4.::X20AI8321_109.AInput[3] AT %IW."X20AI8321_109".AnalogInput03; (*Current 0 to 20 mA / current 4 to 20 mA ; P4 is working with current 4 to 20 mA, resolution 12 bit*)
	Cyclic#4.::X20AI8321_109.AInput[4] AT %IW."X20AI8321_109".AnalogInput04; (*Current 0 to 20 mA / current 4 to 20 mA ; P4 is working with current 4 to 20 mA, resolution 12 bit*)
	Cyclic#4.::X20AI8321_109.AInput[5] AT %IW."X20AI8321_109".AnalogInput05; (*Current 0 to 20 mA / current 4 to 20 mA ; P4 is working with current 4 to 20 mA, resolution 12 bit*)
	Cyclic#4.::X20AI8321_109.AInput[6] AT %IW."X20AI8321_109".AnalogInput06; (*Current 0 to 20 mA / current 4 to 20 mA ; P4 is working with current 4 to 20 mA, resolution 12 bit*)
	Cyclic#4.::X20AI8321_109.AInput[7] AT %IW."X20AI8321_109".AnalogInput07; (*Current 0 to 20 mA / current 4 to 20 mA ; P4 is working with current 4 to 20 mA, resolution 12 bit*)
	Cyclic#4.::X20AI8321_109.AInput[8] AT %IW."X20AI8321_109".AnalogInput08; (*Current 0 to 20 mA / current 4 to 20 mA ; P4 is working with current 4 to 20 mA, resolution 12 bit*)
	Cyclic#4.::X20AI8321_110.AInput[1] AT %IW."X20AI8321_110".AnalogInput01;
	Cyclic#4.::X20AI8321_110.AInput[2] AT %IW."X20AI8321_110".AnalogInput02;
	Cyclic#4.::X20AI8321_110.AInput[3] AT %IW."X20AI8321_110".AnalogInput03;
	Cyclic#4.::X20AI8321_110.AInput[4] AT %IW."X20AI8321_110".AnalogInput04;
	Cyclic#4.::X20AI8321_110.AInput[5] AT %IW."X20AI8321_110".AnalogInput05;
	Cyclic#4.::X20AI8321_110.AInput[6] AT %IW."X20AI8321_110".AnalogInput06;
	Cyclic#4.::X20AI8321_110.AInput[7] AT %IW."X20AI8321_110".AnalogInput07;
	Cyclic#4.::X20AI8321_110.AInput[8] AT %IW."X20AI8321_110".AnalogInput08;
	Cyclic#4.::X20AI8321_109.ModuleOk AT %IX."X20AI8321_109".ModuleOk;
	Cyclic#4.::X20AI8321_110.ModuleOk AT %IX."X20AI8321_110".ModuleOk;
	Cyclic#4.::X20AO4622_111.AOutput[1] AT %QW."X20AO4622_111".AnalogOutput01;
	Cyclic#4.::X20AO4622_111.AOutput[2] AT %QW."X20AO4622_111".AnalogOutput02;
	Cyclic#4.::X20AO4622_111.AOutput[3] AT %QW."X20AO4622_111".AnalogOutput03;
	Cyclic#4.::X20AO4622_111.AOutput[4] AT %QW."X20AO4622_111".AnalogOutput04;
	Cyclic#4.::X20AO4622_112.AOutput[1] AT %QW."X20AO4622_112".AnalogOutput01;
	Cyclic#4.::X20AO4622_112.AOutput[2] AT %QW."X20AO4622_112".AnalogOutput02;
	Cyclic#4.::X20AO4622_112.AOutput[3] AT %QW."X20AO4622_112".AnalogOutput03;
	Cyclic#4.::X20AO4622_112.AOutput[4] AT %QW."X20AO4622_112".AnalogOutput04;
	Cyclic#4.::X20AO4622_113.AOutput[1] AT %QW."X20AO4622_113".AnalogOutput01;
	Cyclic#4.::X20AO4622_113.AOutput[2] AT %QW."X20AO4622_113".AnalogOutput02;
	Cyclic#4.::X20AO4622_113.AOutput[3] AT %QW."X20AO4622_113".AnalogOutput03;
	Cyclic#4.::X20AO4622_113.AOutput[4] AT %QW."X20AO4622_113".AnalogOutput04;
	Cyclic#4.::X20AO4622_111.ModuleOk AT %IX."X20AO4622_111".ModuleOk;
	Cyclic#4.::X20AO4622_112.ModuleOk AT %IX."X20AO4622_112".ModuleOk;
	Cyclic#4.::X20AO4622_113.ModuleOk AT %IX."X20AO4622_113".ModuleOk;
	Cyclic#4.::X20AT4222_114.TempInput[2] AT %IW."X20AT4222_114".Temperature02;
	Cyclic#4.::X20AT4222_114.TempInput[3] AT %IW."X20AT4222_114".Temperature03;
	Cyclic#4.::X20AT4222_114.TempInput[4] AT %IW."X20AT4222_114".Temperature04;
	Cyclic#4.::X20AT4222_114.TempInput[1] AT %IW."X20AT4222_114".Temperature01;
	Cyclic#4.::X20AT4222_114.Status01 AT %IB."X20AT4222_114".StatusInput01;
	Cyclic#4.::X20AT4222_114.ModuleOk AT %IX."X20AT4222_114".ModuleOk;
	Cyclic#4.::X20AT4222_115.ModuleOk AT %IX."X20AT4222_115".ModuleOk;
	Cyclic#4.::X20AT4222_115.TempInput[1] AT %IW."X20AT4222_115".Temperature01;
	Cyclic#4.::X20AT4222_115.TempInput[2] AT %IW."X20AT4222_115".Temperature02;
	Cyclic#4.::X20AT4222_115.TempInput[3] AT %IW."X20AT4222_115".Temperature03;
	Cyclic#4.::X20AT4222_115.TempInput[4] AT %IW."X20AT4222_115".Temperature04;
	Cyclic#4.::X20AT4222_115.Status01 AT %IB."X20AT4222_115".StatusInput01;
	Cyclic#4.::X20AT4222_116.ModuleOk AT %IX."X20AT4222_116".ModuleOk;
	Cyclic#4.::X20AT4222_116.Status01 AT %IB."X20AT4222_116".StatusInput01;
	Cyclic#4.::X20AT4222_116.TempInput[1] AT %IW."X20AT4222_116".Temperature01;
	Cyclic#4.::X20AT4222_116.TempInput[2] AT %IW."X20AT4222_116".Temperature02;
	Cyclic#4.::X20AT4222_116.TempInput[3] AT %IW."X20AT4222_116".Temperature03;
	Cyclic#4.::X20AT4222_116.TempInput[4] AT %IW."X20AT4222_116".Temperature04;
	Cyclic#4.::X20AI8321_110.Status01 AT %IB."X20AI8321_110".StatusInput01;
	Cyclic#4.::X20AI8321_110.Status02 AT %IB."X20AI8321_110".StatusInput02;
	Cyclic#4.::X20AI8321_109.Status01 AT %IB."X20AI8321_109".StatusInput01;
	Cyclic#4.::X20AI8321_109.Status02 AT %IB."X20AI8321_109".StatusInput02;
	Cyclic#1.::SiUnitBK1.ModuleOk AT %IX."SI_unit_BK1".ModuleOk;
	Cyclic#1.::SiUnitBK1.NodeStatus AT %IW."SI_unit_BK1".NodeStatus;
	Cyclic#1.::SiUnitBK1.Input01_08 AT %IB."SI_unit_BK1".ReadInout1hTo8h_6000sub1;
	Cyclic#1.::SiUnitBK1.Input09_16 AT %IB."SI_unit_BK1".ReadInput9hTo16h_6000sub2;
	Cyclic#1.::SiUnitBK1.Input17_24 AT %IB."SI_unit_BK1".ReadInput17hTo24h_6000sub3;
	Cyclic#1.::SiUnitBK1.Input25_32 AT %IB."SI_unit_BK1".ReadInput25hTo32h_6000sub4;
	Cyclic#1.::SiUnitBK1.Output01_08 AT %QB."SI_unit_BK1".WriteOutput1hTo8h_6200sub1;
	Cyclic#1.::SiUnitBK1.Output09_16 AT %QB."SI_unit_BK1".WriteOutput9hTo16h_6200sub2;
	Cyclic#1.::SiUnitBK1.Output17_24 AT %QB."SI_unit_BK1".WriteOutput17hTo24h_6200sub3;
	Cyclic#1.::SiUnitBK1.Output25_32 AT %QB."SI_unit_BK1".WriteOutput25hTo32h_6200sub4;
	Cyclic#1.::SiUnitBK2.ModuleOk AT %IX."SI_unit_BK2".ModuleOk;
	Cyclic#1.::SiUnitBK2.NodeStatus AT %IW."SI_unit_BK2".NodeStatus;
	Cyclic#1.::SiUnitBK2.Input01_08 AT %IB."SI_unit_BK2".ReadInout1hTo8h_6000sub1;
	Cyclic#1.::SiUnitBK2.Input09_16 AT %IB."SI_unit_BK2".ReadInput9hTo16h_6000sub2;
	Cyclic#1.::SiUnitBK2.Input17_24 AT %IB."SI_unit_BK2".ReadInput17hTo24h_6000sub3;
	Cyclic#1.::SiUnitBK2.Input25_32 AT %IB."SI_unit_BK2".ReadInput25hTo32h_6000sub4;
	Cyclic#1.::SiUnitBK2.Output01_08 AT %QB."SI_unit_BK2".WriteOutput1hTo8h_6200sub1;
	Cyclic#1.::SiUnitBK2.Output09_16 AT %QB."SI_unit_BK2".WriteOutput9hTo16h_6200sub2;
	Cyclic#1.::SiUnitBK2.Output17_24 AT %QB."SI_unit_BK2".WriteOutput17hTo24h_6200sub3;
	Cyclic#1.::SiUnitBK2.Output25_32 AT %QB."SI_unit_BK2".WriteOutput25hTo32h_6200sub4;
	Cyclic#4.::X3.DInput[5] AT %IX."X3".DigitalInput05;
	Cyclic#4.::X3.DInput[6] AT %IX."X3".DigitalInput06;
	Cyclic#4.::X3.DInput[7] AT %IX."X3".DigitalInput07;
	Cyclic#4.::X3.DOutput[1] AT %QX."X3".DigitalOutput01;
	Cyclic#4.::X3.DOutput[2] AT %QX."X3".DigitalOutput02;
	Cyclic#4.::X3.DOutput[3] AT %QX."X3".DigitalOutput03;
	Cyclic#4.::X3.DOutput[4] AT %QX."X3".DigitalOutput04;
	Cyclic#4.::X3.DOutput[8] AT %QX."X3".DigitalOutput08;
	Cyclic#4.::X3.DOutput[9] AT %QX."X3".DigitalOutput09;
	Cyclic#4.::X3.DOutput[10] AT %QX."X3".DigitalOutput10;
	Cyclic#4.::X3.DOutput[11] AT %QX."X3".DigitalOutput11;
	Cyclic#4.::X3.DOutput[12] AT %QX."X3".DigitalOutput12;
	Cyclic#4.::X20DOF322_106.ModuleOk AT %IX."X20DOF322_106".ModuleOk;
	Cyclic#4.::X20DOF322_106.DOutput[1] AT %QX."X20DOF322_106".DigitalOutput01;
	Cyclic#4.::X20DOF322_106.DOutput[2] AT %QX."X20DOF322_106".DigitalOutput02;
	Cyclic#4.::X20DOF322_106.DOutput[3] AT %QX."X20DOF322_106".DigitalOutput03;
	Cyclic#4.::X20DOF322_106.DOutput[4] AT %QX."X20DOF322_106".DigitalOutput04;
	Cyclic#4.::X20DOF322_106.DOutput[5] AT %QX."X20DOF322_106".DigitalOutput05;
	Cyclic#4.::X20DOF322_106.DOutput[6] AT %QX."X20DOF322_106".DigitalOutput06;
	Cyclic#4.::X20DOF322_106.DOutput[7] AT %QX."X20DOF322_106".DigitalOutput07;
	Cyclic#4.::X20DOF322_106.DOutput[8] AT %QX."X20DOF322_106".DigitalOutput08;
	Cyclic#4.::X20DOF322_106.DOutput[9] AT %QX."X20DOF322_106".DigitalOutput09;
	Cyclic#4.::X20DOF322_106.DOutput[10] AT %QX."X20DOF322_106".DigitalOutput10;
	Cyclic#4.::X20DOF322_106.DOutput[11] AT %QX."X20DOF322_106".DigitalOutput11;
	Cyclic#4.::X20DOF322_106.DOutput[12] AT %QX."X20DOF322_106".DigitalOutput12;
	Cyclic#4.::X20DOF322_106.DOutput[13] AT %QX."X20DOF322_106".DigitalOutput13;
	Cyclic#4.::X20DOF322_106.DOutput[14] AT %QX."X20DOF322_106".DigitalOutput14;
	Cyclic#4.::X20DOF322_106.DOutput[15] AT %QX."X20DOF322_106".DigitalOutput15;
	Cyclic#4.::X20DOF322_106.DOutput[16] AT %QX."X20DOF322_106".DigitalOutput16;
	Cyclic#4.::X20DOF322_107.ModuleOk AT %IX."X20DOF322_107".ModuleOk;
	Cyclic#4.::X20DOF322_107.DOutput[1] AT %QX."X20DOF322_107".DigitalOutput01;
	Cyclic#4.::X20DOF322_107.DOutput[2] AT %QX."X20DOF322_107".DigitalOutput02;
	Cyclic#4.::X20DOF322_107.DOutput[3] AT %QX."X20DOF322_107".DigitalOutput03;
	Cyclic#4.::X20DOF322_107.DOutput[4] AT %QX."X20DOF322_107".DigitalOutput04;
	Cyclic#4.::X20DOF322_107.DOutput[5] AT %QX."X20DOF322_107".DigitalOutput05;
	Cyclic#4.::X20DOF322_107.DOutput[6] AT %QX."X20DOF322_107".DigitalOutput06;
	Cyclic#4.::X20DOF322_107.DOutput[7] AT %QX."X20DOF322_107".DigitalOutput07;
	Cyclic#4.::X20DOF322_107.DOutput[8] AT %QX."X20DOF322_107".DigitalOutput08;
	Cyclic#4.::X20DOF322_107.DOutput[9] AT %QX."X20DOF322_107".DigitalOutput09;
	Cyclic#4.::X20DOF322_107.DOutput[10] AT %QX."X20DOF322_107".DigitalOutput10;
	Cyclic#4.::X20DOF322_107.DOutput[11] AT %QX."X20DOF322_107".DigitalOutput11;
	Cyclic#4.::X20DOF322_107.DOutput[12] AT %QX."X20DOF322_107".DigitalOutput12;
	Cyclic#4.::X20DOF322_107.DOutput[13] AT %QX."X20DOF322_107".DigitalOutput13;
	Cyclic#4.::X20DOF322_107.DOutput[14] AT %QX."X20DOF322_107".DigitalOutput14;
	Cyclic#4.::X20DOF322_107.DOutput[15] AT %QX."X20DOF322_107".DigitalOutput15;
	Cyclic#4.::X20DOF322_107.DOutput[16] AT %QX."X20DOF322_107".DigitalOutput16;
	Cyclic#4.::X20DOF322_108.ModuleOk AT %IX."X20DOF322_108".ModuleOk;
	Cyclic#4.::X20DOF322_108.DOutput[1] AT %QX."X20DOF322_108".DigitalOutput01;
	Cyclic#4.::X20DOF322_108.DOutput[2] AT %QX."X20DOF322_108".DigitalOutput02;
	Cyclic#4.::X20DOF322_108.DOutput[3] AT %QX."X20DOF322_108".DigitalOutput03;
	Cyclic#4.::X20DOF322_108.DOutput[4] AT %QX."X20DOF322_108".DigitalOutput04;
	Cyclic#4.::X20DOF322_108.DOutput[5] AT %QX."X20DOF322_108".DigitalOutput05;
	Cyclic#4.::X20DOF322_108.DOutput[6] AT %QX."X20DOF322_108".DigitalOutput06;
	Cyclic#4.::X20DOF322_108.DOutput[7] AT %QX."X20DOF322_108".DigitalOutput07;
	Cyclic#4.::X20DOF322_108.DOutput[8] AT %QX."X20DOF322_108".DigitalOutput08;
	Cyclic#4.::X20DOF322_108.DOutput[9] AT %QX."X20DOF322_108".DigitalOutput09;
	Cyclic#4.::X20DOF322_108.DOutput[10] AT %QX."X20DOF322_108".DigitalOutput10;
	Cyclic#4.::X20DOF322_108.DOutput[11] AT %QX."X20DOF322_108".DigitalOutput11;
	Cyclic#4.::X20DOF322_108.DOutput[12] AT %QX."X20DOF322_108".DigitalOutput12;
	Cyclic#4.::X20DOF322_108.DOutput[13] AT %QX."X20DOF322_108".DigitalOutput13;
	Cyclic#4.::X20DOF322_108.DOutput[14] AT %QX."X20DOF322_108".DigitalOutput14;
	Cyclic#4.::X20DOF322_108.DOutput[15] AT %QX."X20DOF322_108".DigitalOutput15;
	Cyclic#4.::X20DOF322_108.DOutput[16] AT %QX."X20DOF322_108".DigitalOutput16;
	Cyclic#4.::X20AI2636_005.ModuleOk AT %IX."X20AI2636_005".ModuleOk;
	Cyclic#4.::X20AI2636_005.AInput[10] AT %IW."X20AI2636_005".PhysCh01Sample10;
	Cyclic#4.::X20AI2636_005.AInput[9] AT %IW."X20AI2636_005".PhysCh01Sample9;
	Cyclic#4.::X20AI2636_005.AInput[8] AT %IW."X20AI2636_005".PhysCh01Sample8;
	Cyclic#4.::X20AI2636_005.AInput[7] AT %IW."X20AI2636_005".PhysCh01Sample7;
	Cyclic#4.::X20AI2636_005.AInput[6] AT %IW."X20AI2636_005".PhysCh01Sample6;
	Cyclic#4.::X20AI2636_005.AInput[5] AT %IW."X20AI2636_005".PhysCh01Sample5;
	Cyclic#4.::X20AI2636_005.AInput[4] AT %IW."X20AI2636_005".PhysCh01Sample4;
	Cyclic#4.::X20AI2636_005.AInput[3] AT %IW."X20AI2636_005".PhysCh01Sample3;
	Cyclic#4.::X20AI2636_005.AInput[2] AT %IW."X20AI2636_005".PhysCh01Sample2;
	Cyclic#4.::X20AI2636_005.AInput[1] AT %IW."X20AI2636_005".PhysCh01Sample1;
	Cyclic#4.::X20DIF371_201.DInput[1] AT %IX."X20DIF371_201".DigitalInput01;
	Cyclic#4.::X20DIF371_201.DInput[2] AT %IX."X20DIF371_201".DigitalInput02;
	Cyclic#4.::X20DIF371_201.DInput[3] AT %IX."X20DIF371_201".DigitalInput03;
	Cyclic#4.::X20DIF371_201.DInput[4] AT %IX."X20DIF371_201".DigitalInput04;
	Cyclic#4.::X20DIF371_201.DInput[5] AT %IX."X20DIF371_201".DigitalInput05;
	Cyclic#4.::X20DIF371_201.DInput[6] AT %IX."X20DIF371_201".DigitalInput06;
	Cyclic#4.::X20DIF371_201.DInput[7] AT %IX."X20DIF371_201".DigitalInput07;
	Cyclic#4.::X20DIF371_201.DInput[8] AT %IX."X20DIF371_201".DigitalInput08;
	Cyclic#4.::X20DIF371_201.DInput[9] AT %IX."X20DIF371_201".DigitalInput09;
	Cyclic#4.::X20DIF371_201.DInput[10] AT %IX."X20DIF371_201".DigitalInput10;
	Cyclic#4.::X20DIF371_202.DInput[1] AT %IX."X20DIF371_202".DigitalInput01;
	Cyclic#4.::X20DIF371_202.DInput[2] AT %IX."X20DIF371_202".DigitalInput02;
	Cyclic#4.::X20DIF371_202.DInput[3] AT %IX."X20DIF371_202".DigitalInput03;
	Cyclic#4.::X20DIF371_202.DInput[4] AT %IX."X20DIF371_202".DigitalInput04;
	Cyclic#4.::X20DIF371_202.DInput[5] AT %IX."X20DIF371_202".DigitalInput05;
	Cyclic#4.::X20DIF371_202.DInput[6] AT %IX."X20DIF371_202".DigitalInput06;
	Cyclic#4.::X20DIF371_202.DInput[7] AT %IX."X20DIF371_202".DigitalInput07;
	Cyclic#4.::X20DIF371_202.DInput[8] AT %IX."X20DIF371_202".DigitalInput08;
	Cyclic#4.::X20DIF371_202.DInput[9] AT %IX."X20DIF371_202".DigitalInput09;
	Cyclic#4.::X20DIF371_202.DInput[10] AT %IX."X20DIF371_202".DigitalInput10;
	Cyclic#4.::X20DIF371_202.DInput[11] AT %IX."X20DIF371_202".DigitalInput11;
	Cyclic#4.::X20DIF371_202.DInput[12] AT %IX."X20DIF371_202".DigitalInput12;
	Cyclic#4.::X20DIF371_202.DInput[13] AT %IX."X20DIF371_202".DigitalInput13;
	Cyclic#4.::X20DIF371_202.DInput[14] AT %IX."X20DIF371_202".DigitalInput14;
	Cyclic#4.::X20DIF371_202.DInput[15] AT %IX."X20DIF371_202".DigitalInput15;
	Cyclic#4.::X20DIF371_202.DInput[16] AT %IX."X20DIF371_202".DigitalInput16;
	Cyclic#4.::X20DIF371_203.DInput[2] AT %IX."X20DIF371_203".DigitalInput02;
	Cyclic#4.::X20DIF371_203.DInput[3] AT %IX."X20DIF371_203".DigitalInput03;
	Cyclic#4.::X20DIF371_203.DInput[4] AT %IX."X20DIF371_203".DigitalInput04;
	Cyclic#4.::X20DIF371_203.DInput[5] AT %IX."X20DIF371_203".DigitalInput05;
	Cyclic#4.::X20DIF371_203.DInput[6] AT %IX."X20DIF371_203".DigitalInput06;
	Cyclic#4.::X20DIF371_203.DInput[7] AT %IX."X20DIF371_203".DigitalInput07;
	Cyclic#4.::X20DIF371_203.DInput[8] AT %IX."X20DIF371_203".DigitalInput08;
	Cyclic#4.::X20DIF371_203.DInput[9] AT %IX."X20DIF371_203".DigitalInput09;
	Cyclic#4.::X20DIF371_203.DInput[10] AT %IX."X20DIF371_203".DigitalInput10;
	Cyclic#4.::X20DIF371_203.DInput[11] AT %IX."X20DIF371_203".DigitalInput11;
	Cyclic#4.::X20DIF371_203.DInput[12] AT %IX."X20DIF371_203".DigitalInput12;
	Cyclic#4.::X20DIF371_203.DInput[13] AT %IX."X20DIF371_203".DigitalInput13;
	Cyclic#4.::X20DIF371_203.DInput[14] AT %IX."X20DIF371_203".DigitalInput14;
	Cyclic#4.::X20DIF371_203.DInput[15] AT %IX."X20DIF371_203".DigitalInput15;
	Cyclic#4.::X20DIF371_203.DInput[16] AT %IX."X20DIF371_203".DigitalInput16;
	Cyclic#4.::X20DIF371_201.ModuleOk AT %IX."X20DIF371_201".ModuleOk;
	Cyclic#4.::X20DIF371_202.ModuleOk AT %IX."X20DIF371_202".ModuleOk;
	Cyclic#4.::X20DIF371_203.ModuleOk AT %IX."X20DIF371_203".ModuleOk;
	Cyclic#4.::X20AI8321_209.AInput[2] AT %IW."X20AI8321_209".AnalogInput02; (*Current 0 to 20 mA / current 4 to 20 mA ; P4 is working with current 4 to 20 mA, resolution 12 bit*)
	Cyclic#4.::X20AI8321_209.AInput[3] AT %IW."X20AI8321_209".AnalogInput03; (*Current 0 to 20 mA / current 4 to 20 mA ; P4 is working with current 4 to 20 mA, resolution 12 bit*)
	Cyclic#4.::X20AI8321_209.AInput[4] AT %IW."X20AI8321_209".AnalogInput04; (*Current 0 to 20 mA / current 4 to 20 mA ; P4 is working with current 4 to 20 mA, resolution 12 bit*)
	Cyclic#4.::X20AI8321_209.AInput[5] AT %IW."X20AI8321_209".AnalogInput05; (*Current 0 to 20 mA / current 4 to 20 mA ; P4 is working with current 4 to 20 mA, resolution 12 bit*)
	Cyclic#4.::X20AI8321_209.AInput[6] AT %IW."X20AI8321_209".AnalogInput06; (*Current 0 to 20 mA / current 4 to 20 mA ; P4 is working with current 4 to 20 mA, resolution 12 bit*)
	Cyclic#4.::X20AI8321_210.AInput[2] AT %IW."X20AI8321_210".AnalogInput02; (*Current 0 to 20 mA / current 4 to 20 mA ; P4 is working with current 4 to 20 mA, resolution 12 bit*)
	Cyclic#4.::X20AI8321_210.AInput[3] AT %IW."X20AI8321_210".AnalogInput03; (*Current 0 to 20 mA / current 4 to 20 mA ; P4 is working with current 4 to 20 mA, resolution 12 bit*)
	Cyclic#4.::X20AI8321_210.AInput[4] AT %IW."X20AI8321_210".AnalogInput04; (*Current 0 to 20 mA / current 4 to 20 mA ; P4 is working with current 4 to 20 mA, resolution 12 bit*)
	Cyclic#4.::X20AI8321_210.AInput[5] AT %IW."X20AI8321_210".AnalogInput05; (*Current 0 to 20 mA / current 4 to 20 mA ; P4 is working with current 4 to 20 mA, resolution 12 bit*)
	Cyclic#4.::X20AI8321_210.AInput[6] AT %IW."X20AI8321_210".AnalogInput06; (*Current 0 to 20 mA / current 4 to 20 mA ; P4 is working with current 4 to 20 mA, resolution 12 bit*)
	Cyclic#4.::X20AI8321_210.AInput[7] AT %IW."X20AI8321_210".AnalogInput07; (*Current 0 to 20 mA / current 4 to 20 mA ; P4 is working with current 4 to 20 mA, resolution 12 bit*)
	Cyclic#4.::X20AI8321_210.AInput[8] AT %IW."X20AI8321_210".AnalogInput08; (*Current 0 to 20 mA / current 4 to 20 mA ; P4 is working with current 4 to 20 mA, resolution 12 bit*)
	Cyclic#4.::X20AI8321_209.ModuleOk AT %IX."X20AI8321_209".ModuleOk;
	Cyclic#4.::X20AI8321_210.ModuleOk AT %IX."X20AI8321_210".ModuleOk;
	Cyclic#4.::X20AO4622_212.AOutput[1] AT %QW."X20AO4622_212".AnalogOutput01;
	Cyclic#4.::X20AO4622_212.AOutput[2] AT %QW."X20AO4622_212".AnalogOutput02;
	Cyclic#4.::X20AO4622_212.AOutput[3] AT %QW."X20AO4622_212".AnalogOutput03;
	Cyclic#4.::X20AO4622_212.AOutput[4] AT %QW."X20AO4622_212".AnalogOutput04;
	Cyclic#4.::X20AO4622_213.AOutput[1] AT %QW."X20AO4622_213".AnalogOutput01;
	Cyclic#4.::X20AO4622_213.AOutput[2] AT %QW."X20AO4622_213".AnalogOutput02;
	Cyclic#4.::X20AO4622_213.AOutput[3] AT %QW."X20AO4622_213".AnalogOutput03;
	Cyclic#4.::X20AO4622_213.AOutput[4] AT %QW."X20AO4622_213".AnalogOutput04;
	Cyclic#4.::X20AO4622_212.ModuleOk AT %IX."X20AO4622_212".ModuleOk;
	Cyclic#4.::X20AO4622_213.ModuleOk AT %IX."X20AO4622_213".ModuleOk;
	Cyclic#4.::X20AT4222_214.TempInput[2] AT %IW."X20AT4222_214".Temperature02;
	Cyclic#4.::X20AT4222_214.TempInput[3] AT %IW."X20AT4222_214".Temperature03;
	Cyclic#4.::X20AT4222_214.TempInput[4] AT %IW."X20AT4222_214".Temperature04;
	Cyclic#4.::X20AT4222_214.TempInput[1] AT %IW."X20AT4222_214".Temperature01;
	Cyclic#4.::X20AT4222_214.Status01 AT %IB."X20AT4222_214".StatusInput01;
	Cyclic#4.::X20AT4222_214.ModuleOk AT %IX."X20AT4222_214".ModuleOk;
	Cyclic#4.::X20AT4222_215.ModuleOk AT %IX."X20AT4222_215".ModuleOk;
	Cyclic#4.::X20AT4222_215.TempInput[1] AT %IW."X20AT4222_215".Temperature01;
	Cyclic#4.::X20AT4222_215.TempInput[2] AT %IW."X20AT4222_215".Temperature02;
	Cyclic#4.::X20AT4222_215.Status01 AT %IB."X20AT4222_215".StatusInput01;
	Cyclic#4.::X20AT4222_216.ModuleOk AT %IX."X20AT4222_216".ModuleOk;
	Cyclic#4.::X20AT4222_216.Status01 AT %IB."X20AT4222_216".StatusInput01;
	Cyclic#4.::X20AT4222_216.TempInput[1] AT %IW."X20AT4222_216".Temperature01;
	Cyclic#4.::X20AT4222_216.TempInput[2] AT %IW."X20AT4222_216".Temperature02;
	Cyclic#4.::X20AT4222_216.TempInput[3] AT %IW."X20AT4222_216".Temperature03;
	Cyclic#4.::X20AT4222_216.TempInput[4] AT %IW."X20AT4222_216".Temperature04;
	Cyclic#4.::X20AI8321_210.Status01 AT %IB."X20AI8321_210".StatusInput01;
	Cyclic#4.::X20AI8321_210.Status02 AT %IB."X20AI8321_210".StatusInput02;
	Cyclic#4.::X20AI8321_209.Status01 AT %IB."X20AI8321_209".StatusInput01;
	Cyclic#4.::X20AI8321_209.Status02 AT %IB."X20AI8321_209".StatusInput02;
	Cyclic#4.::X20DIF371_201.DInput[11] AT %IX."X20DIF371_201".DigitalInput11;
	Cyclic#4.::X20DIF371_201.DInput[12] AT %IX."X20DIF371_201".DigitalInput12;
	Cyclic#4.::X20DIF371_201.DInput[13] AT %IX."X20DIF371_201".DigitalInput13;
	Cyclic#4.::X20DIF371_201.DInput[14] AT %IX."X20DIF371_201".DigitalInput14;
	Cyclic#4.::X20DIF371_201.DInput[15] AT %IX."X20DIF371_201".DigitalInput15;
	Cyclic#4.::X20DIF371_201.DInput[16] AT %IX."X20DIF371_201".DigitalInput16;
	Cyclic#4.::X20DIF371_203.DInput[1] AT %IX."X20DIF371_203".DigitalInput01;
	Cyclic#4.::X20AI8321_209.AInput[1] AT %IW."X20AI8321_209".AnalogInput01; (*Current 0 to 20 mA / current 4 to 20 mA ; P4 is working with current 4 to 20 mA, resolution 12 bit*)
	Cyclic#4.::X20AI8321_209.AInput[7] AT %IW."X20AI8321_209".AnalogInput07; (*Current 0 to 20 mA / current 4 to 20 mA ; P4 is working with current 4 to 20 mA, resolution 12 bit*)
	Cyclic#4.::X20AI8321_209.AInput[8] AT %IW."X20AI8321_209".AnalogInput08; (*Current 0 to 20 mA / current 4 to 20 mA ; P4 is working with current 4 to 20 mA, resolution 12 bit*)
	Cyclic#4.::X20AI8321_210.AInput[1] AT %IW."X20AI8321_210".AnalogInput01; (*Current 0 to 20 mA / current 4 to 20 mA ; P4 is working with current 4 to 20 mA, resolution 12 bit*)
	Cyclic#4.::X20AO4622_211.AOutput[1] AT %QW."X20AO4622_211".AnalogOutput01;
	Cyclic#4.::X20AO4622_211.AOutput[2] AT %QW."X20AO4622_211".AnalogOutput02;
	Cyclic#4.::X20AO4622_211.AOutput[3] AT %QW."X20AO4622_211".AnalogOutput03;
	Cyclic#4.::X20AO4622_211.AOutput[4] AT %QW."X20AO4622_211".AnalogOutput04;
	Cyclic#4.::X20AO4622_211.ModuleOk AT %IX."X20AO4622_211".ModuleOk;
	Cyclic#4.::X20AT4222_215.TempInput[3] AT %IW."X20AT4222_215".Temperature03;
	Cyclic#4.::X20AT4222_215.TempInput[4] AT %IW."X20AT4222_215".Temperature04;
	Cyclic#1.::gIclaNetData[1].xModuleOK AT %IX."ILE1F_BK1".ModuleOk;
	Cyclic#1.::gIclaNetData[1].RPDO4.driveCtrl AT %QB."ILE1F_BK1".Pdo4_driveCtrl_301Esub1;
	Cyclic#1.::gIclaNetData[1].RPDO4.modeCtrl AT %QB."ILE1F_BK1".Pdo4_modeCtrl_301Esub2;
	Cyclic#1.::gIclaNetData[1].TPDO4.modeStat AT %IB."ILE1F_BK1".Pdo4_modeStat_301Esub3;
	Cyclic#1.::gIclaNetData[1].TPDO4.driveStat AT %IW."ILE1F_BK1".Pdo4_driveStat_301Esub4;
	Cyclic#1.::gIclaNetData[1].RPDO4.Ref16 AT %QW."ILE1F_BK1".Pdo4_Ref16_301Esub5;
	Cyclic#1.::gIclaNetData[1].RPDO4.Ref32 AT %QD."ILE1F_BK1".Pdo4_Ref32_301Esub6;
	Cyclic#1.::gIclaNetData[1].TPDO4.Act32 AT %ID."ILE1F_BK1".Pdo4_Act32_301Esub8;
	Cyclic#1.::gIclaNetData[1].TPDO4.Act8 AT %IB."ILE1F_BK1".Pdo4_Act8_301Esub7;
	Cyclic#1.::gIclaNetData[2].xModuleOK AT %IX."ILE1F_BK2".ModuleOk;
	Cyclic#1.::gIclaNetData[2].RPDO4.driveCtrl AT %QB."ILE1F_BK2".Pdo4_driveCtrl_301Esub1;
	Cyclic#1.::gIclaNetData[2].RPDO4.modeCtrl AT %QB."ILE1F_BK2".Pdo4_modeCtrl_301Esub2;
	Cyclic#1.::gIclaNetData[2].TPDO4.modeStat AT %IB."ILE1F_BK2".Pdo4_modeStat_301Esub3;
	Cyclic#1.::gIclaNetData[2].TPDO4.driveStat AT %IW."ILE1F_BK2".Pdo4_driveStat_301Esub4;
	Cyclic#1.::gIclaNetData[2].RPDO4.Ref16 AT %QW."ILE1F_BK2".Pdo4_Ref16_301Esub5;
	Cyclic#1.::gIclaNetData[2].RPDO4.Ref32 AT %QD."ILE1F_BK2".Pdo4_Ref32_301Esub6;
	Cyclic#1.::gIclaNetData[2].TPDO4.Act8 AT %IB."ILE1F_BK2".Pdo4_Act8_301Esub7;
	Cyclic#1.::gIclaNetData[2].TPDO4.Act32 AT %ID."ILE1F_BK2".Pdo4_Act32_301Esub8;
	Cyclic#4.::X20DC4395_104.ModuleOk AT %IX."X20DC4395_104".ModuleOk;
	Cyclic#4.::X20DC4395_104.CountInput[1] AT %IW."X20DC4395_104".EventCounter01;
	Cyclic#4.::X20DC4395_104.CountInput[2] AT %IW."X20DC4395_104".EventCounter02;
	Cyclic#4.::X20DC4395_104.CountInput[3] AT %IW."X20DC4395_104".EventCounter03;
	Cyclic#4.::X20DC4395_104.CountInput[4] AT %IW."X20DC4395_104".EventCounter04;
	Cyclic#4.::X20DC4395_104.CountInput[5] AT %IW."X20DC4395_104".EventCounter05;
	Cyclic#4.::X20DC4395_104.CountInput[6] AT %IW."X20DC4395_104".EventCounter06;
	Cyclic#4.::X20DC4395_104.CountInput[7] AT %IW."X20DC4395_104".EventCounter07;
	Cyclic#4.::X20DC4395_104.CountInput[8] AT %IW."X20DC4395_104".EventCounter08;
	Cyclic#4.::X20DC4395_105.CountInput[1] AT %IW."X20DC4395_105".EventCounter01;
	Cyclic#4.::X20DC4395_105.ModuleOk AT %IX."X20DC4395_105".ModuleOk;
	Cyclic#4.::X20DC4395_105.CountInput[2] AT %IW."X20DC4395_105".EventCounter02;
	Cyclic#4.::X20DC4395_105.CountInput[3] AT %IW."X20DC4395_105".EventCounter03;
	Cyclic#4.::X20DC4395_105.CountInput[4] AT %IW."X20DC4395_105".EventCounter04;
	Cyclic#4.::X20DC4395_105.CountInput[5] AT %IW."X20DC4395_105".EventCounter05;
	Cyclic#4.::X20DC4395_105.CountInput[6] AT %IW."X20DC4395_105".EventCounter06;
	Cyclic#4.::X20DC4395_105.CountInput[7] AT %IW."X20DC4395_105".EventCounter07;
	Cyclic#4.::X20DC4395_105.CountInput[8] AT %IW."X20DC4395_105".EventCounter08;
	Cyclic#4.::X20SO2110_218.DInput[1] AT %IX."X20SO2110_218".PhysicalStateChannel1; (*Read back value of channel Up Down Enable Phys*)
	Cyclic#4.::X20SLX402_006.DOutput[1] AT %QX."X20SC0402".DigitalOutput01; (*Enable Transport signal*)
	Cyclic#4.::X20SLX402_006.DInput[10] AT %IX."X20SC0402".PhysicalStateChannel01;
	Cyclic#4.::X20SO2110_118.DInput[1] AT %IX."X20SO2110_118".PhysicalStateChannel1; (*Read back value of channel SafetyOk means?? *)
	Cyclic#4.::X20SO2110_118.DOutput[1] AT %QX."X20SO2110_118".DigitalOutput01;
	Cyclic#4.::X20SO2110_118.DOutput[2] AT %QX."X20SO2110_118".DigitalOutput02;
	Cyclic#4.::X20SO2110_218.DOutput[1] AT %QX."X20SO2110_218".DigitalOutput01;
	Cyclic#4.::X20SO2110_218.DOutput[2] AT %QX."X20SO2110_218".DigitalOutput02;
	Cyclic#4.::X20SLX402_006.DInput[1] AT %IX."X20SC0402".SafeDigitalInput01;
	Cyclic#4.::X20SI8110_217.DInput[1] AT %IX."X20SI8110_217".SafeDigitalInput01;
	Cyclic#4.::X20SI8110_217.DInput[3] AT %IX."X20SI8110_217".SafeDigitalInput03;
	Cyclic#4.::X20SI8110_217.DInput[2] AT %IX."X20SI8110_217".SafeDigitalInput02;
	Cyclic#4.::X20SI8110_217.DInput[4] AT %IX."X20SI8110_217".SafeDigitalInput04;
	Cyclic#4.::X20SI8110_217.DInput[5] AT %IX."X20SI8110_217".SafeDigitalInput05;
	Cyclic#4.::X20SI8110_217.DInput[6] AT %IX."X20SI8110_217".SafeDigitalInput06;
	Cyclic#4.::X20SI8110_217.DInput[7] AT %IX."X20SI8110_217".SafeDigitalInput07;
	Cyclic#4.::X20DOF322_207.DOutput[9] AT %QX."X20DOF322_207".DigitalOutput09;
	Cyclic#4.::X20DOF322_207.DOutput[10] AT %QX."X20DOF322_207".DigitalOutput10;
	Cyclic#4.::X20DOF322_207.DOutput[11] AT %QX."X20DOF322_207".DigitalOutput11;
	Cyclic#4.::X20DOF322_207.DOutput[12] AT %QX."X20DOF322_207".DigitalOutput12;
	Cyclic#4.::X20DOF322_207.DOutput[13] AT %QX."X20DOF322_207".DigitalOutput13;
	Cyclic#4.::X20DOF322_207.DOutput[14] AT %QX."X20DOF322_207".DigitalOutput14;
	Cyclic#4.::X20DOF322_207.DOutput[15] AT %QX."X20DOF322_207".DigitalOutput15;
	Cyclic#4.::X20DOF322_207.DOutput[16] AT %QX."X20DOF322_207".DigitalOutput16;
	Cyclic#4.::X20DOF322_208.DOutput[1] AT %QX."X20DOF322_208".DigitalOutput01;
	Cyclic#4.::X20DOF322_208.DOutput[2] AT %QX."X20DOF322_208".DigitalOutput02;
	Cyclic#4.::X20DOF322_208.DOutput[3] AT %QX."X20DOF322_208".DigitalOutput03;
	Cyclic#4.::X20DOF322_208.DOutput[4] AT %QX."X20DOF322_208".DigitalOutput04;
	Cyclic#4.::X20DOF322_208.DOutput[5] AT %QX."X20DOF322_208".DigitalOutput05;
	Cyclic#4.::X20DOF322_208.DOutput[6] AT %QX."X20DOF322_208".DigitalOutput06;
	Cyclic#4.::X20DOF322_208.DOutput[7] AT %QX."X20DOF322_208".DigitalOutput07;
	Cyclic#4.::X20DOF322_208.DOutput[8] AT %QX."X20DOF322_208".DigitalOutput08;
	Cyclic#4.::X20DOF322_208.DOutput[9] AT %QX."X20DOF322_208".DigitalOutput09;
	Cyclic#4.::X20DOF322_208.DOutput[10] AT %QX."X20DOF322_208".DigitalOutput10;
	Cyclic#4.::X20DOF322_208.DOutput[11] AT %QX."X20DOF322_208".DigitalOutput11;
	Cyclic#4.::X20DOF322_208.DOutput[12] AT %QX."X20DOF322_208".DigitalOutput12;
	Cyclic#4.::X20DOF322_208.DOutput[13] AT %QX."X20DOF322_208".DigitalOutput13;
	Cyclic#4.::X20DOF322_208.DOutput[14] AT %QX."X20DOF322_208".DigitalOutput14;
	Cyclic#4.::X20DOF322_208.DOutput[15] AT %QX."X20DOF322_208".DigitalOutput15;
	Cyclic#4.::X20DOF322_208.DOutput[16] AT %QX."X20DOF322_208".DigitalOutput16;
	Cyclic#4.::X20DOF322_206.DOutput[1] AT %QX."X20DOF322_206".DigitalOutput01;
	Cyclic#4.::X20DOF322_206.DOutput[2] AT %QX."X20DOF322_206".DigitalOutput02;
	Cyclic#4.::X20DOF322_206.DOutput[3] AT %QX."X20DOF322_206".DigitalOutput03;
	Cyclic#4.::X20DOF322_206.DOutput[4] AT %QX."X20DOF322_206".DigitalOutput04;
	Cyclic#4.::X20DOF322_206.DOutput[5] AT %QX."X20DOF322_206".DigitalOutput05;
	Cyclic#4.::X20DOF322_206.DOutput[6] AT %QX."X20DOF322_206".DigitalOutput06;
	Cyclic#4.::X20DOF322_206.DOutput[7] AT %QX."X20DOF322_206".DigitalOutput07;
	Cyclic#4.::X20DOF322_206.DOutput[8] AT %QX."X20DOF322_206".DigitalOutput08;
	Cyclic#4.::X20DOF322_206.DOutput[9] AT %QX."X20DOF322_206".DigitalOutput09;
	Cyclic#4.::X20DOF322_206.DOutput[10] AT %QX."X20DOF322_206".DigitalOutput10;
	Cyclic#4.::X20DOF322_206.DOutput[11] AT %QX."X20DOF322_206".DigitalOutput11;
	Cyclic#4.::X20DOF322_206.DOutput[12] AT %QX."X20DOF322_206".DigitalOutput12;
	Cyclic#4.::X20DOF322_206.DOutput[13] AT %QX."X20DOF322_206".DigitalOutput13;
	Cyclic#4.::X20DOF322_206.DOutput[14] AT %QX."X20DOF322_206".DigitalOutput14;
	Cyclic#4.::X20DOF322_206.DOutput[15] AT %QX."X20DOF322_206".DigitalOutput15;
	Cyclic#4.::X20DOF322_206.DOutput[16] AT %QX."X20DOF322_206".DigitalOutput16;
	Cyclic#4.::X20DOF322_208.ModuleOk AT %IX."X20DOF322_208".ModuleOk;
	Cyclic#4.::X20DOF322_207.ModuleOk AT %IX."X20DOF322_207".ModuleOk;
	Cyclic#4.::X20DOF322_206.ModuleOk AT %IX."X20DOF322_206".ModuleOk;
	Cyclic#4.::X20DC4395_205.ModuleOk AT %IX."X20DC4395_205".ModuleOk;
	Cyclic#4.::X20DC4395_204.CountInput[1] AT %IW."X20DC4395_204".EventCounter01;
	Cyclic#4.::X20DC4395_204.CountInput[2] AT %IW."X20DC4395_204".EventCounter02;
	Cyclic#4.::X20DC4395_204.CountInput[3] AT %IW."X20DC4395_204".EventCounter03;
	Cyclic#4.::X20DC4395_204.CountInput[4] AT %IW."X20DC4395_204".EventCounter04;
	Cyclic#4.::X20DC4395_204.CountInput[5] AT %IW."X20DC4395_204".EventCounter05;
	Cyclic#4.::X20DC4395_204.CountInput[6] AT %IW."X20DC4395_204".EventCounter06;
	Cyclic#4.::X20DC4395_204.CountInput[7] AT %IW."X20DC4395_204".EventCounter07;
	Cyclic#4.::X20DC4395_204.CountInput[8] AT %IW."X20DC4395_204".EventCounter08;
	Cyclic#4.::X20DC4395_204.ModuleOk AT %IX."X20DC4395_204".ModuleOk;
	Cyclic#4.::X20DC4395_205.CountInput[1] AT %IW."X20DC4395_205".EventCounter01;
	Cyclic#4.::X20DC4395_205.CountInput[2] AT %IW."X20DC4395_205".EventCounter02;
	Cyclic#4.::X20DC4395_205.CountInput[3] AT %IW."X20DC4395_205".EventCounter03;
	Cyclic#4.::X20DC4395_205.CountInput[4] AT %IW."X20DC4395_205".EventCounter04;
	Cyclic#4.::X20DC4395_205.CountInput[5] AT %IW."X20DC4395_205".EventCounter05;
	Cyclic#4.::X20DC4395_205.CountInput[6] AT %IW."X20DC4395_205".EventCounter06;
	Cyclic#4.::X20DC4395_205.CountInput[7] AT %IW."X20DC4395_205".EventCounter07;
	Cyclic#4.::X20DC4395_205.CountInput[8] AT %IW."X20DC4395_205".EventCounter08;
	Cyclic#4.::X20AI2636_005.DInput[1] AT %IX."X20AI2636_005".Channel01Error;
	Cyclic#4.::X20AI2636_005.DOutput[1] AT %QX."X20AI2636_005".AckChannel01Error;
	Cyclic#4.::X20AI2636_005.AInput[11] AT %IW."X20AI2636_005".PhysCh01Sample11;
	Cyclic#4.::X20AI2636_005.AInput[12] AT %IW."X20AI2636_005".PhysCh01Sample12;
	Cyclic#4.::X20DIF371_030.DInput[1] AT %IX."X20DIF371_030".DigitalInput01;
	Cyclic#4.::X20DIF371_030.DInput[2] AT %IX."X20DIF371_030".DigitalInput02;
	Cyclic#4.::X20DIF371_030.DInput[3] AT %IX."X20DIF371_030".DigitalInput03;
	Cyclic#4.::X20DIF371_030.DInput[4] AT %IX."X20DIF371_030".DigitalInput04;
	Cyclic#4.::X20DIF371_030.DInput[5] AT %IX."X20DIF371_030".DigitalInput05;
	Cyclic#4.::X20DIF371_030.DInput[6] AT %IX."X20DIF371_030".DigitalInput06;
	Cyclic#4.::X20DIF371_030.DInput[7] AT %IX."X20DIF371_030".DigitalInput07;
	Cyclic#4.::X20DIF371_030.DInput[8] AT %IX."X20DIF371_030".DigitalInput08;
	Cyclic#4.::X20DIF371_030.DInput[9] AT %IX."X20DIF371_030".DigitalInput09;
	Cyclic#4.::X20DIF371_030.DInput[10] AT %IX."X20DIF371_030".DigitalInput10;
	Cyclic#4.::X20DIF371_030.DInput[11] AT %IX."X20DIF371_030".DigitalInput11;
	Cyclic#4.::X20DIF371_030.DInput[12] AT %IX."X20DIF371_030".DigitalInput12;
	Cyclic#4.::X20DIF371_030.DInput[13] AT %IX."X20DIF371_030".DigitalInput13;
	Cyclic#4.::X20DIF371_030.DInput[14] AT %IX."X20DIF371_030".DigitalInput14;
	Cyclic#4.::X20DIF371_030.DInput[15] AT %IX."X20DIF371_030".DigitalInput15;
	Cyclic#4.::X20DIF371_030.DInput[16] AT %IX."X20DIF371_030".DigitalInput16;
	Cyclic#4.::X20DIF371_030.ModuleOk AT %IX."X20DIF371_030".ModuleOk;
	Cyclic#4.::X20SI8110_217.DInput[8] AT %IX."X20SI8110_217".SafeDigitalInput08;
	Cyclic#4.::X20SI8110_117.DInput[1] AT %IX."X20SI8110_117".SafeDigitalInput01;
	Cyclic#4.::X20SI8110_117.DInput[2] AT %IX."X20SI8110_117".SafeDigitalInput02;
	Cyclic#4.::X20SI8110_117.DInput[3] AT %IX."X20SI8110_117".SafeDigitalInput03;
	Cyclic#4.::X20SI8110_117.DInput[4] AT %IX."X20SI8110_117".SafeDigitalInput04;
	Cyclic#4.::X20SI8110_117.DInput[5] AT %IX."X20SI8110_117".SafeDigitalInput05;
	Cyclic#4.::X20SI8110_117.DInput[6] AT %IX."X20SI8110_117".SafeDigitalInput06;
	Cyclic#4.::X20SI8110_117.DInput[7] AT %IX."X20SI8110_117".SafeDigitalInput07;
	Cyclic#4.::X20DOF322_207.DOutput[1] AT %QX."X20DOF322_207".DigitalOutput01;
	Cyclic#4.::X20DOF322_207.DOutput[2] AT %QX."X20DOF322_207".DigitalOutput02;
	Cyclic#4.::X20DOF322_207.DOutput[3] AT %QX."X20DOF322_207".DigitalOutput03;
	Cyclic#4.::X20DOF322_207.DOutput[4] AT %QX."X20DOF322_207".DigitalOutput04;
	Cyclic#4.::X20DOF322_207.DOutput[5] AT %QX."X20DOF322_207".DigitalOutput05;
	Cyclic#4.::X20DOF322_207.DOutput[6] AT %QX."X20DOF322_207".DigitalOutput06;
	Cyclic#4.::X20DOF322_207.DOutput[7] AT %QX."X20DOF322_207".DigitalOutput07;
	Cyclic#4.::X20DOF322_207.DOutput[8] AT %QX."X20DOF322_207".DigitalOutput08;
	Cyclic#1.::gAxisStepper[1].DrvIf.iLifeCnt AT %IB."X20SM1436_007".LifeCnt;
	Cyclic#1.::gAxisStepper[1].DrvIf.iDrvOK AT %IX."X20SM1436_007".DrvOk01;
	Cyclic#1.::gAxisStepper[1].DrvIf.oBoostCurrent AT %QX."X20SM1436_007".BoostCurrent01;
	Cyclic#1.::gAxisStepper[1].DrvIf.oStandStillCurrent AT %QX."X20SM1436_007".StandstillCurrent01;
	Cyclic#1.::gAxisStepper[1].DrvIf.oSetTime AT %QW."X20SM1436_007".SetTime01;
	Cyclic#1.::gAxisStepper[1].DiDoIf.iLifeCntDriveEnable AT %IB."X20SM1436_007".LifeCnt;
	Cyclic#1.::gAxisStepper[1].DiDoIf.iLifeCntDriveReady AT %IB."X20SM1436_007".LifeCnt;
	Cyclic#1.::gAxisStepper[1].DiDoIf.iDriveReady AT %IX."X20SM1436_007".DrvOk01;
	Cyclic#1.::gAxisStepper[1].EncIf1.iLifeCnt AT %IB."X20SM1436_007".LifeCnt;
	Cyclic#1.::gAxisStepper[1].EncIf1.iEncOK AT %IX."X20SM1436_007".EncOk01;
	Cyclic#1.::gAxisStepper[1].EncIf1.iActPos AT %IW."X20SM1436_007".ActPos01;
	Cyclic#1.::gAxisStepper[1].EncIf1.iRefPulsePos AT %IW."X20SM1436_007".RefPulsePos01;
	Cyclic#1.::gAxisStepper[1].EncIf1.iRefPulseCnt AT %IB."X20SM1436_007".RefPulseCnt01;
	Cyclic#1.::gAxisStepper[1].EncIf1.iActTime AT %IW."X20SM1436_007".ActTime01;
	Cyclic#1.::X20SM1436_007.ModuleOk AT %IX."X20SM1436_007".ModuleOk;
	Cyclic#1.::gAxisStepper[1].DiDoIf.oDriveEnable AT %QX."X20SM1436_007".DriveEnable01;
	Cyclic#1.::gAxisStepper[1].MotorStep0 AT %QW."X20SM1436_007".Motor1Step0;
	Cyclic#1.::gAxisStepper[2].DrvIf.iLifeCnt AT %IB."X20SM1436_008".LifeCnt;
	Cyclic#1.::gAxisStepper[2].DrvIf.iDrvOK AT %IX."X20SM1436_008".DrvOk01;
	Cyclic#1.::gAxisStepper[2].DrvIf.oBoostCurrent AT %QX."X20SM1436_008".BoostCurrent01;
	Cyclic#1.::gAxisStepper[2].DrvIf.oStandStillCurrent AT %QX."X20SM1436_008".StandstillCurrent01;
	Cyclic#1.::gAxisStepper[2].DrvIf.oSetTime AT %QW."X20SM1436_008".SetTime01;
	Cyclic#1.::gAxisStepper[2].MotorStep0 AT %QW."X20SM1436_008".Motor1Step0;
	Cyclic#1.::gAxisStepper[2].DiDoIf.iLifeCntDriveEnable AT %IB."X20SM1436_008".LifeCnt;
	Cyclic#1.::gAxisStepper[2].DiDoIf.iLifeCntDriveReady AT %IB."X20SM1436_008".LifeCnt;
	Cyclic#1.::gAxisStepper[2].DiDoIf.iDriveReady AT %IX."X20SM1436_008".DrvOk01;
	Cyclic#1.::gAxisStepper[2].DiDoIf.oDriveEnable AT %QX."X20SM1436_008".DriveEnable01;
	Cyclic#1.::gAxisStepper[2].EncIf1.iLifeCnt AT %IB."X20SM1436_008".LifeCnt;
	Cyclic#1.::gAxisStepper[2].EncIf1.iEncOK AT %IX."X20SM1436_008".EncOk01;
	Cyclic#1.::gAxisStepper[2].EncIf1.iActPos AT %IW."X20SM1436_008".ActPos01;
	Cyclic#1.::gAxisStepper[2].EncIf1.iRefPulsePos AT %IW."X20SM1436_008".RefPulsePos01;
	Cyclic#1.::gAxisStepper[2].EncIf1.iRefPulseCnt AT %IB."X20SM1436_008".RefPulseCnt01;
	Cyclic#1.::gAxisStepper[2].EncIf1.iActTime AT %IW."X20SM1436_008".ActTime01;
	Cyclic#1.X20SM1436_008.ModuleOk AT %IX."X20SM1436_008".ModuleOk;
	Cyclic#4.::X20AI2636_005.AInput[13] AT %IW."X20AI2636_005".PhysCh01Sample13;
	::X20DIF371_003.ModuleOk AT %IX."X20DIF371_003".ModuleOk;
	::X20SLX402_006.ModuleOk AT %IX."X20SC0402".ModuleOk;
	::X20SI8110_117.ModuleOk AT %IX."X20SI8110_117".ModuleOk;
	::X20SO2110_118.ModuleOk AT %IX."X20SO2110_118".ModuleOk;
	::X20SI8110_217.ModuleOk AT %IX."X20SI8110_217".ModuleOk;
	::X20SO2110_218.ModuleOk AT %IX."X20SO2110_218".ModuleOk;
END_VAR
```

### Acp10map.ncm - X20CP1382/Motion/Acp10map.ncm
```
NcMapping (NcSwId=Acp10, DisabledNodesAreHidden=False)
  NcObject gAxis01 (ModuleId=8V1045.00-2_BELT, Type=ncAXIS, Channel=1, AcoposSimulation=Off, InitParameter=BeltI, AcoposParameter=BeltA, Disabled=FALSE, ModuleDisabled=FALSE)
  NcObject 8V1045.00-2_ncV_AXIS1 (ModuleId=8V1045.00-2_BELT, Type=ncV_AXIS, Channel=1, Disabled=TRUE, ModuleDisabled=FALSE)
  NcObject gAxis21 (ModuleId=8V1016.50-2_BK1, Type=ncAXIS, Channel=1, AcoposSimulation=Off, InitParameter=BK1_i, AcoposParameter=BK1_a, Disabled=FALSE, ModuleDisabled=FALSE)
  NcObject gAxis121 (ModuleId=8V1016.50-2_BK2, Type=ncAXIS, Channel=1, AcoposSimulation=Off, InitParameter=BK1_i, AcoposParameter=BK1_a, Disabled=FALSE, ModuleDisabled=FALSE)
  NcObject 8V1016.50-2_ncV_AXIS1 (ModuleId=8V1016.50-2_BK2, Type=ncV_AXIS, Channel=1, Disabled=TRUE, ModuleDisabled=FALSE)
  NcObject 8V1016.50-2_ncV_AXIS1 (ModuleId=8V1016.50-2_BK1, Type=ncV_AXIS, Channel=1, Disabled=TRUE, ModuleDisabled=FALSE)
  NcObject gAxisStp01 (ModuleId=X20SM1436_007, ModuleAddress=SDC_IF1.ST1, Type=ncAXIS, Channel=1, AcoposSimulation=Off, InitParameter=SM_i, AcoposParameter=SM_a, AdditionalData=SDC_AX_HwPv="gAxisStepper[1].HW", Disabled=FALSE, ModuleDisabled=FALSE)
  NcObject gAxisStp02 (ModuleId=X20SM1436_008, ModuleAddress=SDC_IF1.ST2, Type=ncAXIS, Channel=1, AcoposSimulation=Off, InitParameter=SM_i, AcoposParameter=SM_a, AdditionalData=SDC_AX_HwPv="gAxisStepper[2].HW", Disabled=FALSE, ModuleDisabled=FALSE)
```

## Configuration Dryer

CPU X20CP0483, AutomationRuntime S4.93, Build 4.1.2, Safety 0.0
